// TIA Portal V20 export
FUNCTION_BLOCK "Sequence_2_SideTapeAttachment"   // FB32852, LAD
TITLE = Sequence
// Sequence template programmend in ladder logic
// stored: IsIECCheckEnabled true, MemoryReserve 100, Namespace Unit1.Em4, SetENOAutomatically true
   VAR_INPUT
      unitStatus { ExternalAccessible := 'False'; ExternalVisible := 'False'; ExternalWritable := 'False'} : "LAF_typeUnitStatus";   // Current unit status o be used in this EM
   END_VAR
   VAR
      instSequenceLADControl { ExternalAccessible := 'False'; ExternalVisible := 'False'; ExternalWritable := 'False'} : "LAF_ControlLadSequence";
      instSequenceLADStatus { ExternalAccessible := 'False'; ExternalVisible := 'False'; ExternalWritable := 'False'} : "LAF_StatusLadSequence";
      statTonTime { ExternalAccessible := 'False'; ExternalVisible := 'False'; ExternalWritable := 'False'} : Array[0..9999] of TON_TIME;
   END_VAR
   VAR_TEMP
      tempCustomerAction : Bool;   // Placeholder for possible actions
      tempDo_nothing_and_wait_for_init : Bool;   // Placeholder for doing nothing
      tempSafeStateCondition : Bool;   // Temp Condition for the equipment module to be in a safe state
   END_VAR
   VAR CONSTANT
      delayTime : Time := T#100ms;
      STEP_IDLE : DInt := 1;
      JOB_1_STEP_1 : DInt := 101;
      JOB_1_STEP_10 : DInt := 110;
      JOB_1_STEP_11 : DInt := 111;
      JOB_1_STEP_20 : DInt := 120;
      JOB_1_STEP_30 : DInt := 130;
      JOB_1_STEP_31 : DInt := 131;
      JOB_1_STEP_32 : DInt := 132;
      JOB_1_STEP_33 : DInt := 133;
      JOB_1_STEP_34 : DInt := 134;
      JOB_1_STEP_40 : DInt := 140;
      JOB_1_STEP_41 : DInt := 141;
      JOB_1_STEP_42 : DInt := 142;
      JOB_1_STEP_43 : DInt := 143;
      JOB_1_STEP_44 : DInt := 144;
      JOB_1_STEP_80 : DInt := 180;
      JOB_1_STEP_81 : DInt := 181;
      JOB_1_STEP_90 : DInt := 190;
      JOB_3_STEP_1 : DInt := 301;
      JOB_3_STEP_10 : DInt := 310;
      JOB_3_STEP_20 : DInt := 320;
      JOB_3_STEP_21 : DInt := 321;
      JOB_3_STEP_30 : DInt := 330;
      JOB_3_STEP_31 : DInt := 331;
      JOB_3_STEP_40 : DInt := 340;
      JOB_3_STEP_41 : DInt := 341;
      JOB_3_STEP_70 : DInt := 370;
      JOB_3_STEP_80 : DInt := 380;
      JOB_3_STEP_90 : DInt := 390;
      JOB_2_STEP_1 : DInt := 201;
      JOB_2_STEP_10 : DInt := 210;
      JOB_2_STEP_20 : DInt := 220;
      JOB_2_STEP_21 : DInt := 221;
      JOB_2_STEP_30 : DInt := 230;
      JOB_2_STEP_31 : DInt := 231;
      JOB_2_STEP_40 : DInt := 240;
      JOB_2_STEP_41 : DInt := 241;
      JOB_2_STEP_70 : DInt := 270;
      JOB_2_STEP_80 : DInt := 280;
      JOB_2_STEP_90 : DInt := 290;
      JOB_4_STEP_1 : DInt := 401;
      JOB_4_STEP_10 : DInt := 410;
      JOB_4_STEP_20 : DInt := 420;
      JOB_4_STEP_21 : DInt := 421;
      JOB_4_STEP_22 : DInt := 422;
      JOB_4_STEP_30 : DInt := 430;
      JOB_4_STEP_31 : DInt := 431;
      JOB_4_STEP_80 : DInt := 480;
      JOB_4_STEP_90 : DInt := 490;
      JOB_5_STEP_1 : DInt := 501;
      JOB_5_STEP_10 : DInt := 510;
      JOB_5_STEP_20 : DInt := 520;
      JOB_5_STEP_21 : DInt := 521;
      JOB_5_STEP_22 : DInt := 522;
      JOB_5_STEP_30 : DInt := 530;
      JOB_5_STEP_31 : DInt := 531;
      JOB_5_STEP_80 : DInt := 580;
      JOB_5_STEP_90 : DInt := 590;
      JOB_6_STEP_1 : DInt := 601;
      JOB_6_STEP_10 : DInt := 610;
      JOB_6_STEP_20 : DInt := 620;
      JOB_6_STEP_21 : DInt := 621;
      JOB_6_STEP_22 : DInt := 622;
      JOB_6_STEP_30 : DInt := 630;
      JOB_6_STEP_31 : DInt := 631;
      JOB_6_STEP_80 : DInt := 680;
      JOB_6_STEP_90 : DInt := 690;
      JOB_7_STEP_1 : DInt := 701;
      JOB_7_STEP_10 : DInt := 710;
      JOB_7_STEP_20 : DInt := 720;
      JOB_7_STEP_21 : DInt := 721;
      JOB_7_STEP_22 : DInt := 722;
      JOB_7_STEP_30 : DInt := 730;
      JOB_7_STEP_31 : DInt := 731;
      JOB_7_STEP_80 : DInt := 780;
      JOB_7_STEP_90 : DInt := 790;
      JOB_8_STEP_1 : DInt := 801;
      JOB_8_STEP_10 : DInt := 810;
      JOB_8_STEP_11 : DInt := 811;
      JOB_8_STEP_12 : DInt := 812;
      JOB_8_STEP_13 : DInt := 813;
      JOB_8_STEP_14 : DInt := 814;
      JOB_8_STEP_15 : DInt := 815;
      JOB_8_STEP_16 : DInt := 816;
      JOB_8_STEP_17 : DInt := 817;
      JOB_8_STEP_20 : DInt := 820;
      JOB_8_STEP_21 : DInt := 821;
      JOB_8_STEP_22 : DInt := 822;
      JOB_8_STEP_23 : DInt := 823;
      JOB_8_STEP_24 : DInt := 824;
      JOB_8_STEP_25 : DInt := 825;
      JOB_8_STEP_26 : DInt := 826;
      JOB_8_STEP_27 : DInt := 827;
      JOB_8_STEP_30 : DInt := 830;
      JOB_8_STEP_31 : DInt := 831;
      JOB_8_STEP_60 : DInt := 860;
      JOB_8_STEP_70 : DInt := 880;
      JOB_8_STEP_80 : DInt := 890;
      STEP_IMMEDIATE_STOP : DInt := 9001;   // Step executed when an immediate stop command is triggered for the sequence (i.e. when unit is in state aborting)
      TO_DO_INSERT_ACTIONS_HERE : Bool := TRUE;   // Template : Add actions
      TO_DO_INSERT_CONDITION_FOR_TRANSITION_HERE : Bool := TRUE;   // Template : Add conditions
   END_VAR
   VAR_TEMP   // added for the SCL form of the ladder/FBD networks
      _w1 : Bool;
      _w2 : Bool;
   END_VAR
BEGIN

REGION Network 1: BLOCK INFO HEADER
   // (company) / (C) Copyright (year)
   // ---------------------------------------------------------------------------------
   // Title:                             (Title of this block)
   // Comment/Function: (that is implemented in the block)
   // Library/Family:           (that the source is dedicated to)
   // Author:                        (department / person in charge / contact)
   // Target System:          (test system with FW version)
   // Engineering:              TIA Portal (SW version)
   // Restrictions:               (OB types, etc.)
   // Requirements:           (hardware, technological package, etc.)
   // ---------------------------------------------------------------------------------
   // Change log table:
   // Version          | Date             | Signature      | Expert in charge  | Changes applied ------------------------|----------------------|-------------------------|--------------------------------|-----------------------
   // 001.000.000 | yyyy-mm-dd | 0x00000000 | (name of expert) | First released version
END_REGION

REGION Network 2: DESCRIPTION
   // This is a template block provided by the Automation Framework. It can be used to create an own project.
   // The Block Info Header is prepared to put in your own data.
   // Description of the block could be added here and the docu created by Code2Docu.
END_REGION

REGION Network 3: *************** CONTROL **********************
END_REGION

REGION Network 4: Sequence Control ("Enter your Sequins number here")
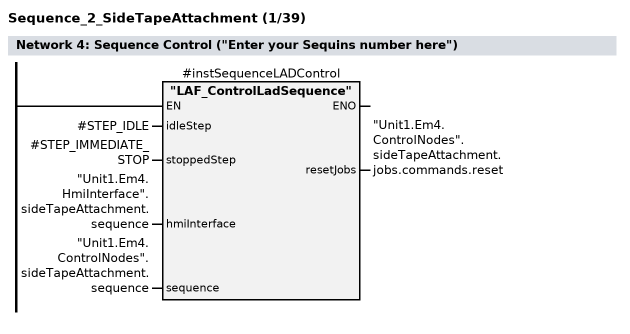
   RUNG wire#powerrail
      #instSequenceLADControl(idleStep := #STEP_IDLE, stoppedStep := #STEP_IMMEDIATE_STOP, hmiInterface := "Unit1.Em4.HmiInterface".sideTapeAttachment.sequence, sequence := "Unit1.Em4.ControlNodes".sideTapeAttachment.sequence, resetJobs => "Unit1.Em4.ControlNodes".sideTapeAttachment.jobs.commands.reset)
   END_RUNG
   // the same network as SCL:
   #instSequenceLADControl(idleStep := #STEP_IDLE,   // "LAF_ControlLadSequence"
                           stoppedStep := #STEP_IMMEDIATE_STOP,
                           hmiInterface := "Unit1.Em4.HmiInterface".sideTapeAttachment.sequence,
                           sequence := "Unit1.Em4.ControlNodes".sideTapeAttachment.sequence,
                           resetJobs => "Unit1.Em4.ControlNodes".sideTapeAttachment.jobs.commands.reset);
END_REGION

REGION Network 5: Step IDLE
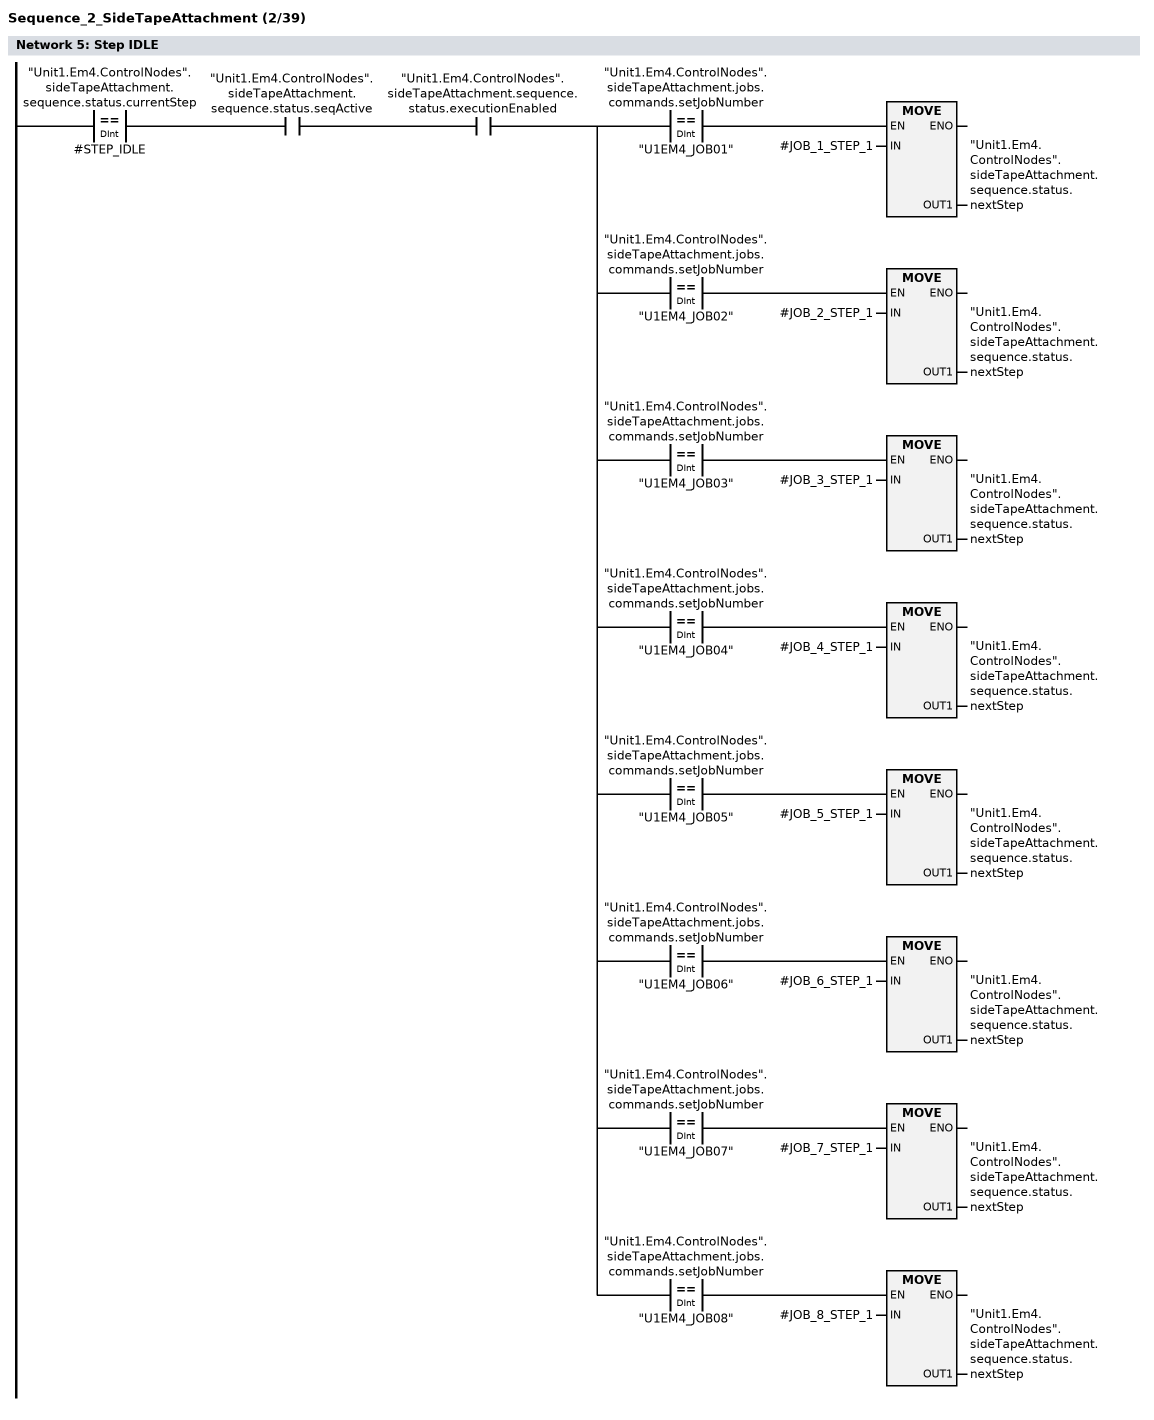
   RUNG wire#powerrail
      { S7_Templates := "SrcType := DInt" } EQ_Contact(in1 := "Unit1.Em4.ControlNodes".sideTapeAttachment.sequence.status.currentStep, in2 := #STEP_IDLE)
      Contact( "Unit1.Em4.ControlNodes".sideTapeAttachment.sequence.status.seqActive )
      Contact( "Unit1.Em4.ControlNodes".sideTapeAttachment.sequence.status.executionEnabled )
      wire#w1
      { S7_Templates := "SrcType := DInt" } EQ_Contact(in1 := "Unit1.Em4.ControlNodes".sideTapeAttachment.jobs.commands.setJobNumber, in2 := "U1EM4_JOB01")
      Move(in := #JOB_1_STEP_1, out1 => "Unit1.Em4.ControlNodes".sideTapeAttachment.sequence.status.nextStep)
   END_RUNG
   RUNG wire#w1
      { S7_Templates := "SrcType := DInt" } EQ_Contact(in1 := "Unit1.Em4.ControlNodes".sideTapeAttachment.jobs.commands.setJobNumber, in2 := "U1EM4_JOB02")
      Move(in := #JOB_2_STEP_1, out1 => "Unit1.Em4.ControlNodes".sideTapeAttachment.sequence.status.nextStep)
   END_RUNG
   RUNG wire#w1
      { S7_Templates := "SrcType := DInt" } EQ_Contact(in1 := "Unit1.Em4.ControlNodes".sideTapeAttachment.jobs.commands.setJobNumber, in2 := "U1EM4_JOB03")
      Move(in := #JOB_3_STEP_1, out1 => "Unit1.Em4.ControlNodes".sideTapeAttachment.sequence.status.nextStep)
   END_RUNG
   RUNG wire#w1
      { S7_Templates := "SrcType := DInt" } EQ_Contact(in1 := "Unit1.Em4.ControlNodes".sideTapeAttachment.jobs.commands.setJobNumber, in2 := "U1EM4_JOB04")
      Move(in := #JOB_4_STEP_1, out1 => "Unit1.Em4.ControlNodes".sideTapeAttachment.sequence.status.nextStep)
   END_RUNG
   RUNG wire#w1
      { S7_Templates := "SrcType := DInt" } EQ_Contact(in1 := "Unit1.Em4.ControlNodes".sideTapeAttachment.jobs.commands.setJobNumber, in2 := "U1EM4_JOB05")
      Move(in := #JOB_5_STEP_1, out1 => "Unit1.Em4.ControlNodes".sideTapeAttachment.sequence.status.nextStep)
   END_RUNG
   RUNG wire#w1
      { S7_Templates := "SrcType := DInt" } EQ_Contact(in1 := "Unit1.Em4.ControlNodes".sideTapeAttachment.jobs.commands.setJobNumber, in2 := "U1EM4_JOB06")
      Move(in := #JOB_6_STEP_1, out1 => "Unit1.Em4.ControlNodes".sideTapeAttachment.sequence.status.nextStep)
   END_RUNG
   RUNG wire#w1
      { S7_Templates := "SrcType := DInt" } EQ_Contact(in1 := "Unit1.Em4.ControlNodes".sideTapeAttachment.jobs.commands.setJobNumber, in2 := "U1EM4_JOB07")
      Move(in := #JOB_7_STEP_1, out1 => "Unit1.Em4.ControlNodes".sideTapeAttachment.sequence.status.nextStep)
   END_RUNG
   RUNG wire#w1
      { S7_Templates := "SrcType := DInt" } EQ_Contact(in1 := "Unit1.Em4.ControlNodes".sideTapeAttachment.jobs.commands.setJobNumber, in2 := "U1EM4_JOB08")
      Move(in := #JOB_8_STEP_1, out1 => "Unit1.Em4.ControlNodes".sideTapeAttachment.sequence.status.nextStep)
   END_RUNG
   // the same network as SCL:
   #_w1 := ("Unit1.Em4.ControlNodes".sideTapeAttachment.sequence.status.currentStep = #STEP_IDLE) AND "Unit1.Em4.ControlNodes".sideTapeAttachment.sequence.status.seqActive AND "Unit1.Em4.ControlNodes".sideTapeAttachment.sequence.status.executionEnabled;
   IF #_w1 AND ("Unit1.Em4.ControlNodes".sideTapeAttachment.jobs.commands.setJobNumber = "U1EM4_JOB01") THEN
       "Unit1.Em4.ControlNodes".sideTapeAttachment.sequence.status.nextStep := #JOB_1_STEP_1;
   END_IF;
   IF #_w1 AND ("Unit1.Em4.ControlNodes".sideTapeAttachment.jobs.commands.setJobNumber = "U1EM4_JOB02") THEN
       "Unit1.Em4.ControlNodes".sideTapeAttachment.sequence.status.nextStep := #JOB_2_STEP_1;
   END_IF;
   IF #_w1 AND ("Unit1.Em4.ControlNodes".sideTapeAttachment.jobs.commands.setJobNumber = "U1EM4_JOB03") THEN
       "Unit1.Em4.ControlNodes".sideTapeAttachment.sequence.status.nextStep := #JOB_3_STEP_1;
   END_IF;
   IF #_w1 AND ("Unit1.Em4.ControlNodes".sideTapeAttachment.jobs.commands.setJobNumber = "U1EM4_JOB04") THEN
       "Unit1.Em4.ControlNodes".sideTapeAttachment.sequence.status.nextStep := #JOB_4_STEP_1;
   END_IF;
   IF #_w1 AND ("Unit1.Em4.ControlNodes".sideTapeAttachment.jobs.commands.setJobNumber = "U1EM4_JOB05") THEN
       "Unit1.Em4.ControlNodes".sideTapeAttachment.sequence.status.nextStep := #JOB_5_STEP_1;
   END_IF;
   IF #_w1 AND ("Unit1.Em4.ControlNodes".sideTapeAttachment.jobs.commands.setJobNumber = "U1EM4_JOB06") THEN
       "Unit1.Em4.ControlNodes".sideTapeAttachment.sequence.status.nextStep := #JOB_6_STEP_1;
   END_IF;
   IF #_w1 AND ("Unit1.Em4.ControlNodes".sideTapeAttachment.jobs.commands.setJobNumber = "U1EM4_JOB07") THEN
       "Unit1.Em4.ControlNodes".sideTapeAttachment.sequence.status.nextStep := #JOB_7_STEP_1;
   END_IF;
   IF #_w1 AND ("Unit1.Em4.ControlNodes".sideTapeAttachment.jobs.commands.setJobNumber = "U1EM4_JOB08") THEN
       "Unit1.Em4.ControlNodes".sideTapeAttachment.sequence.status.nextStep := #JOB_8_STEP_1;
   END_IF;
END_REGION

REGION Network 6: ******************** JOB[1] EM HOMING ********************
END_REGION

REGION Network 7: Step[101] : JOB[1] Condition
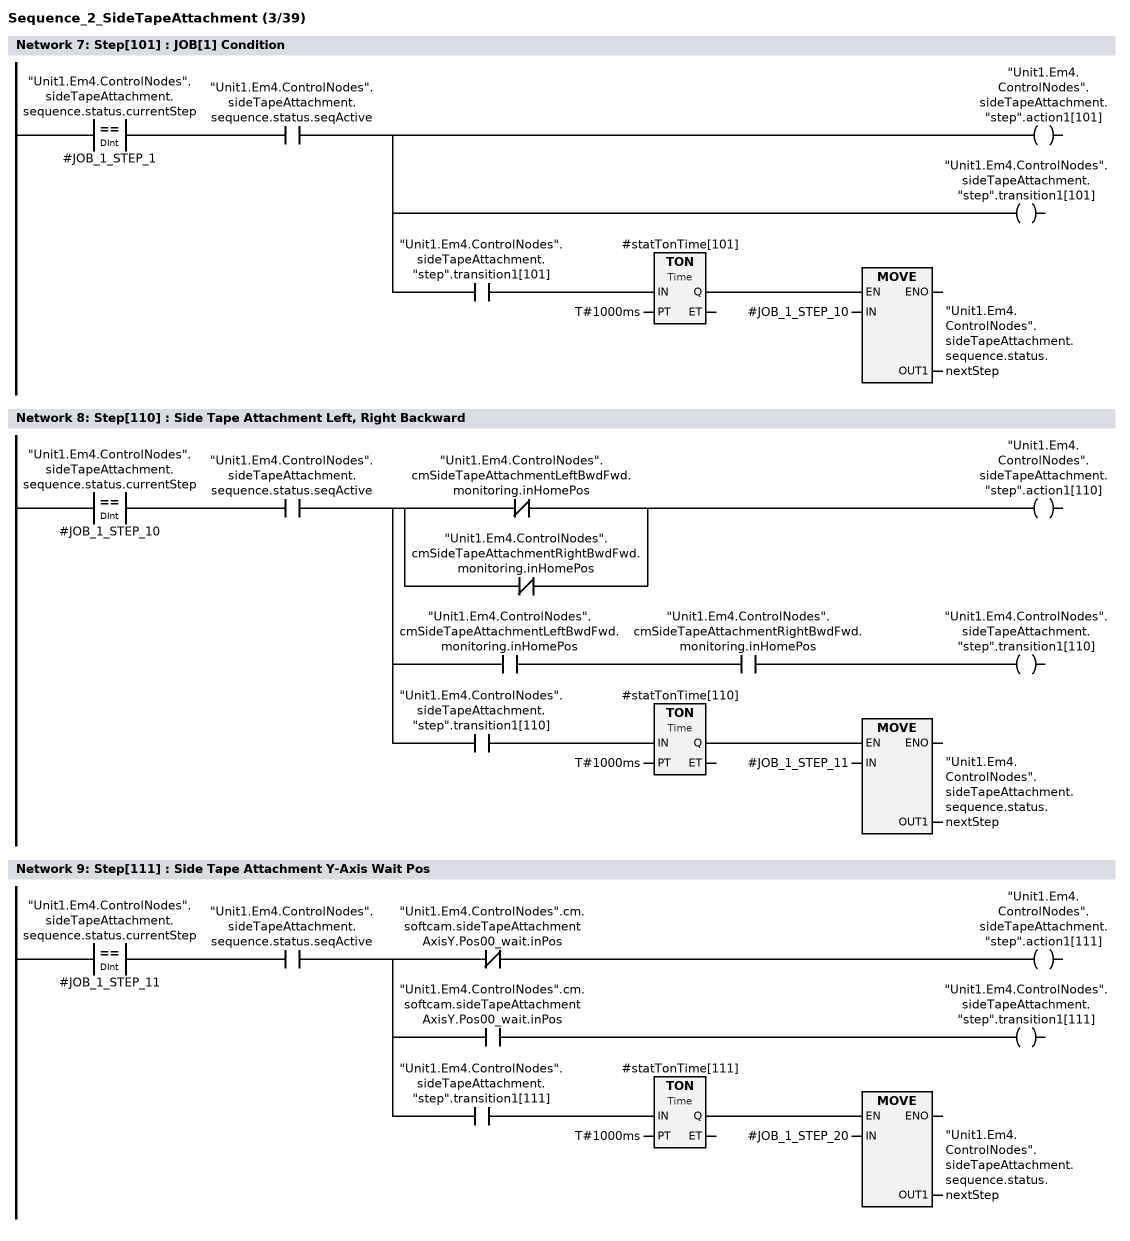
   RUNG wire#powerrail
      { S7_Templates := "SrcType := DInt" } EQ_Contact(in1 := "Unit1.Em4.ControlNodes".sideTapeAttachment.sequence.status.currentStep, in2 := #JOB_1_STEP_1)
      Contact( "Unit1.Em4.ControlNodes".sideTapeAttachment.sequence.status.seqActive )
      wire#w1
      Coil( "Unit1.Em4.ControlNodes".sideTapeAttachment."step".action1[101] )
   END_RUNG
   RUNG wire#w1
      Coil( "Unit1.Em4.ControlNodes".sideTapeAttachment."step".transition1[101] )
   END_RUNG
   RUNG wire#w1
      Contact( "Unit1.Em4.ControlNodes".sideTapeAttachment."step".transition1[101] )
      { S7_Templates := "time_type := Time" } #statTonTime[101].TON(pt := T#1000ms, et =>)
      Move(in := #JOB_1_STEP_10, out1 => "Unit1.Em4.ControlNodes".sideTapeAttachment.sequence.status.nextStep)
   END_RUNG
   // the same network as SCL:
   "Unit1.Em4.ControlNodes".sideTapeAttachment."step".action1[101] := ("Unit1.Em4.ControlNodes".sideTapeAttachment.sequence.status.currentStep = #JOB_1_STEP_1) AND "Unit1.Em4.ControlNodes".sideTapeAttachment.sequence.status.seqActive;
   "Unit1.Em4.ControlNodes".sideTapeAttachment."step".transition1[101] := ("Unit1.Em4.ControlNodes".sideTapeAttachment.sequence.status.currentStep = #JOB_1_STEP_1) AND "Unit1.Em4.ControlNodes".sideTapeAttachment.sequence.status.seqActive;
   #statTonTime[101].TON(IN := ("Unit1.Em4.ControlNodes".sideTapeAttachment.sequence.status.currentStep = #JOB_1_STEP_1) AND "Unit1.Em4.ControlNodes".sideTapeAttachment.sequence.status.seqActive AND "Unit1.Em4.ControlNodes".sideTapeAttachment."step".transition1[101],
                         PT := T#1000ms);
   IF #statTonTime[101].Q THEN
       "Unit1.Em4.ControlNodes".sideTapeAttachment.sequence.status.nextStep := #JOB_1_STEP_10;
   END_IF;
END_REGION

REGION Network 8: Step[110] : Side Tape Attachment Left, Right Backward
   RUNG wire#powerrail
      { S7_Templates := "SrcType := DInt" } EQ_Contact(in1 := "Unit1.Em4.ControlNodes".sideTapeAttachment.sequence.status.currentStep, in2 := #JOB_1_STEP_10)
      Contact( "Unit1.Em4.ControlNodes".sideTapeAttachment.sequence.status.seqActive )
      wire#w1
      I_Contact( "Unit1.Em4.ControlNodes".cmSideTapeAttachmentLeftBwdFwd.monitoring.inHomePos )
      wire#w2
      Coil( "Unit1.Em4.ControlNodes".sideTapeAttachment."step".action1[110] )
   END_RUNG
   RUNG wire#w1
      I_Contact( "Unit1.Em4.ControlNodes".cmSideTapeAttachmentRightBwdFwd.monitoring.inHomePos )
   END_RUNG wire#w2
   RUNG wire#w1
      Contact( "Unit1.Em4.ControlNodes".cmSideTapeAttachmentLeftBwdFwd.monitoring.inHomePos )
      Contact( "Unit1.Em4.ControlNodes".cmSideTapeAttachmentRightBwdFwd.monitoring.inHomePos )
      Coil( "Unit1.Em4.ControlNodes".sideTapeAttachment."step".transition1[110] )
   END_RUNG
   RUNG wire#w1
      Contact( "Unit1.Em4.ControlNodes".sideTapeAttachment."step".transition1[110] )
      { S7_Templates := "time_type := Time" } #statTonTime[110].TON(pt := T#1000ms, et =>)
      Move(in := #JOB_1_STEP_11, out1 => "Unit1.Em4.ControlNodes".sideTapeAttachment.sequence.status.nextStep)
   END_RUNG
   // the same network as SCL:
   #_w1 := ("Unit1.Em4.ControlNodes".sideTapeAttachment.sequence.status.currentStep = #JOB_1_STEP_10) AND "Unit1.Em4.ControlNodes".sideTapeAttachment.sequence.status.seqActive;
   "Unit1.Em4.ControlNodes".sideTapeAttachment."step".action1[110] := #_w1 AND (NOT "Unit1.Em4.ControlNodes".cmSideTapeAttachmentLeftBwdFwd.monitoring.inHomePos OR NOT "Unit1.Em4.ControlNodes".cmSideTapeAttachmentRightBwdFwd.monitoring.inHomePos);
   "Unit1.Em4.ControlNodes".sideTapeAttachment."step".transition1[110] := #_w1 AND "Unit1.Em4.ControlNodes".cmSideTapeAttachmentLeftBwdFwd.monitoring.inHomePos AND "Unit1.Em4.ControlNodes".cmSideTapeAttachmentRightBwdFwd.monitoring.inHomePos;
   #statTonTime[110].TON(IN := #_w1 AND "Unit1.Em4.ControlNodes".sideTapeAttachment."step".transition1[110],
                         PT := T#1000ms);
   IF #statTonTime[110].Q THEN
       "Unit1.Em4.ControlNodes".sideTapeAttachment.sequence.status.nextStep := #JOB_1_STEP_11;
   END_IF;
END_REGION

REGION Network 9: Step[111] : Side Tape Attachment Y-Axis Wait Pos
   RUNG wire#powerrail
      { S7_Templates := "SrcType := DInt" } EQ_Contact(in1 := "Unit1.Em4.ControlNodes".sideTapeAttachment.sequence.status.currentStep, in2 := #JOB_1_STEP_11)
      Contact( "Unit1.Em4.ControlNodes".sideTapeAttachment.sequence.status.seqActive )
      wire#w1
      I_Contact( "Unit1.Em4.ControlNodes".cm.softcam.sideTapeAttachmentAxisY.Pos00_wait.inPos )
      Coil( "Unit1.Em4.ControlNodes".sideTapeAttachment."step".action1[111] )
   END_RUNG
   RUNG wire#w1
      Contact( "Unit1.Em4.ControlNodes".cm.softcam.sideTapeAttachmentAxisY.Pos00_wait.inPos )
      Coil( "Unit1.Em4.ControlNodes".sideTapeAttachment."step".transition1[111] )
   END_RUNG
   RUNG wire#w1
      Contact( "Unit1.Em4.ControlNodes".sideTapeAttachment."step".transition1[111] )
      { S7_Templates := "time_type := Time" } #statTonTime[111].TON(pt := T#1000ms, et =>)
      Move(in := #JOB_1_STEP_20, out1 => "Unit1.Em4.ControlNodes".sideTapeAttachment.sequence.status.nextStep)
   END_RUNG
   // the same network as SCL:
   #_w1 := ("Unit1.Em4.ControlNodes".sideTapeAttachment.sequence.status.currentStep = #JOB_1_STEP_11) AND "Unit1.Em4.ControlNodes".sideTapeAttachment.sequence.status.seqActive;
   "Unit1.Em4.ControlNodes".sideTapeAttachment."step".action1[111] := #_w1 AND NOT "Unit1.Em4.ControlNodes".cm.softcam.sideTapeAttachmentAxisY.Pos00_wait.inPos;
   "Unit1.Em4.ControlNodes".sideTapeAttachment."step".transition1[111] := #_w1 AND "Unit1.Em4.ControlNodes".cm.softcam.sideTapeAttachmentAxisY.Pos00_wait.inPos;
   #statTonTime[111].TON(IN := #_w1 AND "Unit1.Em4.ControlNodes".sideTapeAttachment."step".transition1[111],
                         PT := T#1000ms);
   IF #statTonTime[111].Q THEN
       "Unit1.Em4.ControlNodes".sideTapeAttachment.sequence.status.nextStep := #JOB_1_STEP_20;
   END_IF;
END_REGION

REGION Network 10: Step[120] : Side Tape Attachment Bottom Forward
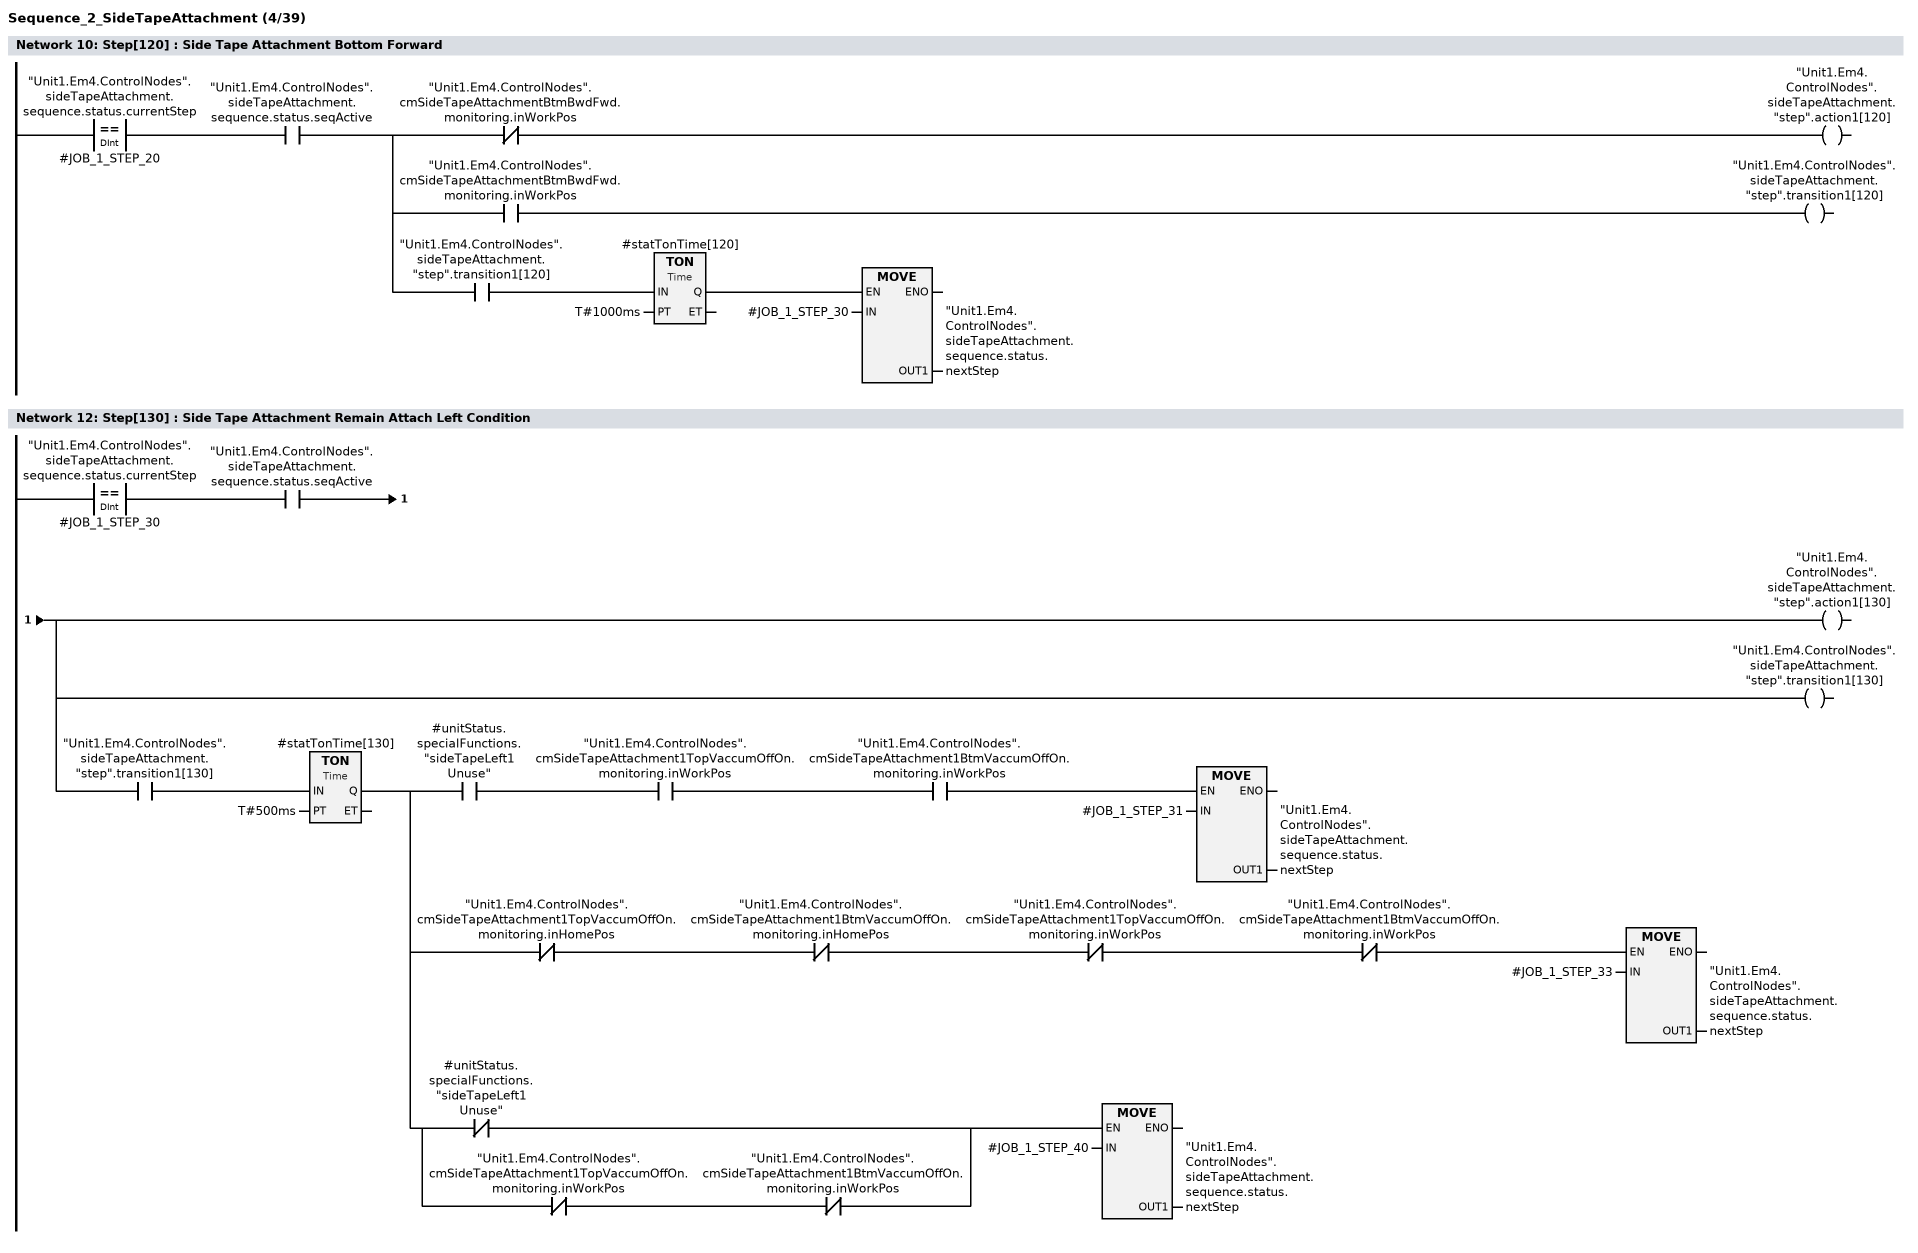
   RUNG wire#powerrail
      { S7_Templates := "SrcType := DInt" } EQ_Contact(in1 := "Unit1.Em4.ControlNodes".sideTapeAttachment.sequence.status.currentStep, in2 := #JOB_1_STEP_20)
      Contact( "Unit1.Em4.ControlNodes".sideTapeAttachment.sequence.status.seqActive )
      wire#w1
      I_Contact( "Unit1.Em4.ControlNodes".cmSideTapeAttachmentBtmBwdFwd.monitoring.inWorkPos )
      Coil( "Unit1.Em4.ControlNodes".sideTapeAttachment."step".action1[120] )
   END_RUNG
   RUNG wire#w1
      Contact( "Unit1.Em4.ControlNodes".cmSideTapeAttachmentBtmBwdFwd.monitoring.inWorkPos )
      Coil( "Unit1.Em4.ControlNodes".sideTapeAttachment."step".transition1[120] )
   END_RUNG
   RUNG wire#w1
      Contact( "Unit1.Em4.ControlNodes".sideTapeAttachment."step".transition1[120] )
      { S7_Templates := "time_type := Time" } #statTonTime[120].TON(pt := T#1000ms, et =>)
      Move(in := #JOB_1_STEP_30, out1 => "Unit1.Em4.ControlNodes".sideTapeAttachment.sequence.status.nextStep)
   END_RUNG
   // the same network as SCL:
   #_w1 := ("Unit1.Em4.ControlNodes".sideTapeAttachment.sequence.status.currentStep = #JOB_1_STEP_20) AND "Unit1.Em4.ControlNodes".sideTapeAttachment.sequence.status.seqActive;
   "Unit1.Em4.ControlNodes".sideTapeAttachment."step".action1[120] := #_w1 AND NOT "Unit1.Em4.ControlNodes".cmSideTapeAttachmentBtmBwdFwd.monitoring.inWorkPos;
   "Unit1.Em4.ControlNodes".sideTapeAttachment."step".transition1[120] := #_w1 AND "Unit1.Em4.ControlNodes".cmSideTapeAttachmentBtmBwdFwd.monitoring.inWorkPos;
   #statTonTime[120].TON(IN := #_w1 AND "Unit1.Em4.ControlNodes".sideTapeAttachment."step".transition1[120],
                         PT := T#1000ms);
   IF #statTonTime[120].Q THEN
       "Unit1.Em4.ControlNodes".sideTapeAttachment.sequence.status.nextStep := #JOB_1_STEP_30;
   END_IF;
END_REGION

REGION Network 11: ******************** STEP[130~134] SIDE TAPE ATTACHMENT LEFT REMAIN ATTACH ********************
END_REGION

REGION Network 12: Step[130] : Side Tape Attachment Remain Attach Left Condition
   RUNG wire#powerrail
      { S7_Templates := "SrcType := DInt" } EQ_Contact(in1 := "Unit1.Em4.ControlNodes".sideTapeAttachment.sequence.status.currentStep, in2 := #JOB_1_STEP_30)
      Contact( "Unit1.Em4.ControlNodes".sideTapeAttachment.sequence.status.seqActive )
      wire#w1
      Coil( "Unit1.Em4.ControlNodes".sideTapeAttachment."step".action1[130] )
   END_RUNG
   RUNG wire#w1
      Coil( "Unit1.Em4.ControlNodes".sideTapeAttachment."step".transition1[130] )
   END_RUNG
   RUNG wire#w1
      Contact( "Unit1.Em4.ControlNodes".sideTapeAttachment."step".transition1[130] )
      { S7_Templates := "time_type := Time" } #statTonTime[130].TON(pt := T#500ms, et =>)
      wire#w2
      Contact( #unitStatus.specialFunctions."sideTapeLeft1 Unuse" )
      Contact( "Unit1.Em4.ControlNodes".cmSideTapeAttachment1TopVaccumOffOn.monitoring.inWorkPos )
      Contact( "Unit1.Em4.ControlNodes".cmSideTapeAttachment1BtmVaccumOffOn.monitoring.inWorkPos )
      Move(in := #JOB_1_STEP_31, out1 => "Unit1.Em4.ControlNodes".sideTapeAttachment.sequence.status.nextStep)
   END_RUNG
   RUNG wire#w2
      I_Contact( "Unit1.Em4.ControlNodes".cmSideTapeAttachment1TopVaccumOffOn.monitoring.inHomePos )
      I_Contact( "Unit1.Em4.ControlNodes".cmSideTapeAttachment1BtmVaccumOffOn.monitoring.inHomePos )
      I_Contact( "Unit1.Em4.ControlNodes".cmSideTapeAttachment1TopVaccumOffOn.monitoring.inWorkPos )
      I_Contact( "Unit1.Em4.ControlNodes".cmSideTapeAttachment1BtmVaccumOffOn.monitoring.inWorkPos )
      Move(in := #JOB_1_STEP_33, out1 => "Unit1.Em4.ControlNodes".sideTapeAttachment.sequence.status.nextStep)
   END_RUNG
   RUNG wire#w2
      I_Contact( #unitStatus.specialFunctions."sideTapeLeft1 Unuse" )
      wire#w3
      Move(in := #JOB_1_STEP_40, out1 => "Unit1.Em4.ControlNodes".sideTapeAttachment.sequence.status.nextStep)
   END_RUNG
   RUNG wire#w2
      I_Contact( "Unit1.Em4.ControlNodes".cmSideTapeAttachment1TopVaccumOffOn.monitoring.inWorkPos )
      I_Contact( "Unit1.Em4.ControlNodes".cmSideTapeAttachment1BtmVaccumOffOn.monitoring.inWorkPos )
   END_RUNG wire#w3
   // the same network as SCL:
   "Unit1.Em4.ControlNodes".sideTapeAttachment."step".action1[130] := ("Unit1.Em4.ControlNodes".sideTapeAttachment.sequence.status.currentStep = #JOB_1_STEP_30) AND "Unit1.Em4.ControlNodes".sideTapeAttachment.sequence.status.seqActive;
   "Unit1.Em4.ControlNodes".sideTapeAttachment."step".transition1[130] := ("Unit1.Em4.ControlNodes".sideTapeAttachment.sequence.status.currentStep = #JOB_1_STEP_30) AND "Unit1.Em4.ControlNodes".sideTapeAttachment.sequence.status.seqActive;
   #statTonTime[130].TON(IN := ("Unit1.Em4.ControlNodes".sideTapeAttachment.sequence.status.currentStep = #JOB_1_STEP_30) AND "Unit1.Em4.ControlNodes".sideTapeAttachment.sequence.status.seqActive AND "Unit1.Em4.ControlNodes".sideTapeAttachment."step".transition1[130],
                         PT := T#500ms);
   IF #statTonTime[130].Q AND #unitStatus.specialFunctions."sideTapeLeft1 Unuse" AND "Unit1.Em4.ControlNodes".cmSideTapeAttachment1TopVaccumOffOn.monitoring.inWorkPos AND "Unit1.Em4.ControlNodes".cmSideTapeAttachment1BtmVaccumOffOn.monitoring.inWorkPos THEN
       "Unit1.Em4.ControlNodes".sideTapeAttachment.sequence.status.nextStep := #JOB_1_STEP_31;
   END_IF;
   IF #statTonTime[130].Q AND NOT "Unit1.Em4.ControlNodes".cmSideTapeAttachment1TopVaccumOffOn.monitoring.inHomePos AND NOT "Unit1.Em4.ControlNodes".cmSideTapeAttachment1BtmVaccumOffOn.monitoring.inHomePos AND NOT "Unit1.Em4.ControlNodes".cmSideTapeAttachment1TopVaccumOffOn.monitoring.inWorkPos AND NOT "Unit1.Em4.ControlNodes".cmSideTapeAttachment1BtmVaccumOffOn.monitoring.inWorkPos THEN
       "Unit1.Em4.ControlNodes".sideTapeAttachment.sequence.status.nextStep := #JOB_1_STEP_33;
   END_IF;
   IF #statTonTime[130].Q AND (NOT #unitStatus.specialFunctions."sideTapeLeft1 Unuse" OR (NOT "Unit1.Em4.ControlNodes".cmSideTapeAttachment1TopVaccumOffOn.monitoring.inWorkPos AND NOT "Unit1.Em4.ControlNodes".cmSideTapeAttachment1BtmVaccumOffOn.monitoring.inWorkPos)) THEN
       "Unit1.Em4.ControlNodes".sideTapeAttachment.sequence.status.nextStep := #JOB_1_STEP_40;
   END_IF;
END_REGION

REGION Network 13: Step[131] : Side Tape Attachment X-Axis Remain Attach Left Position
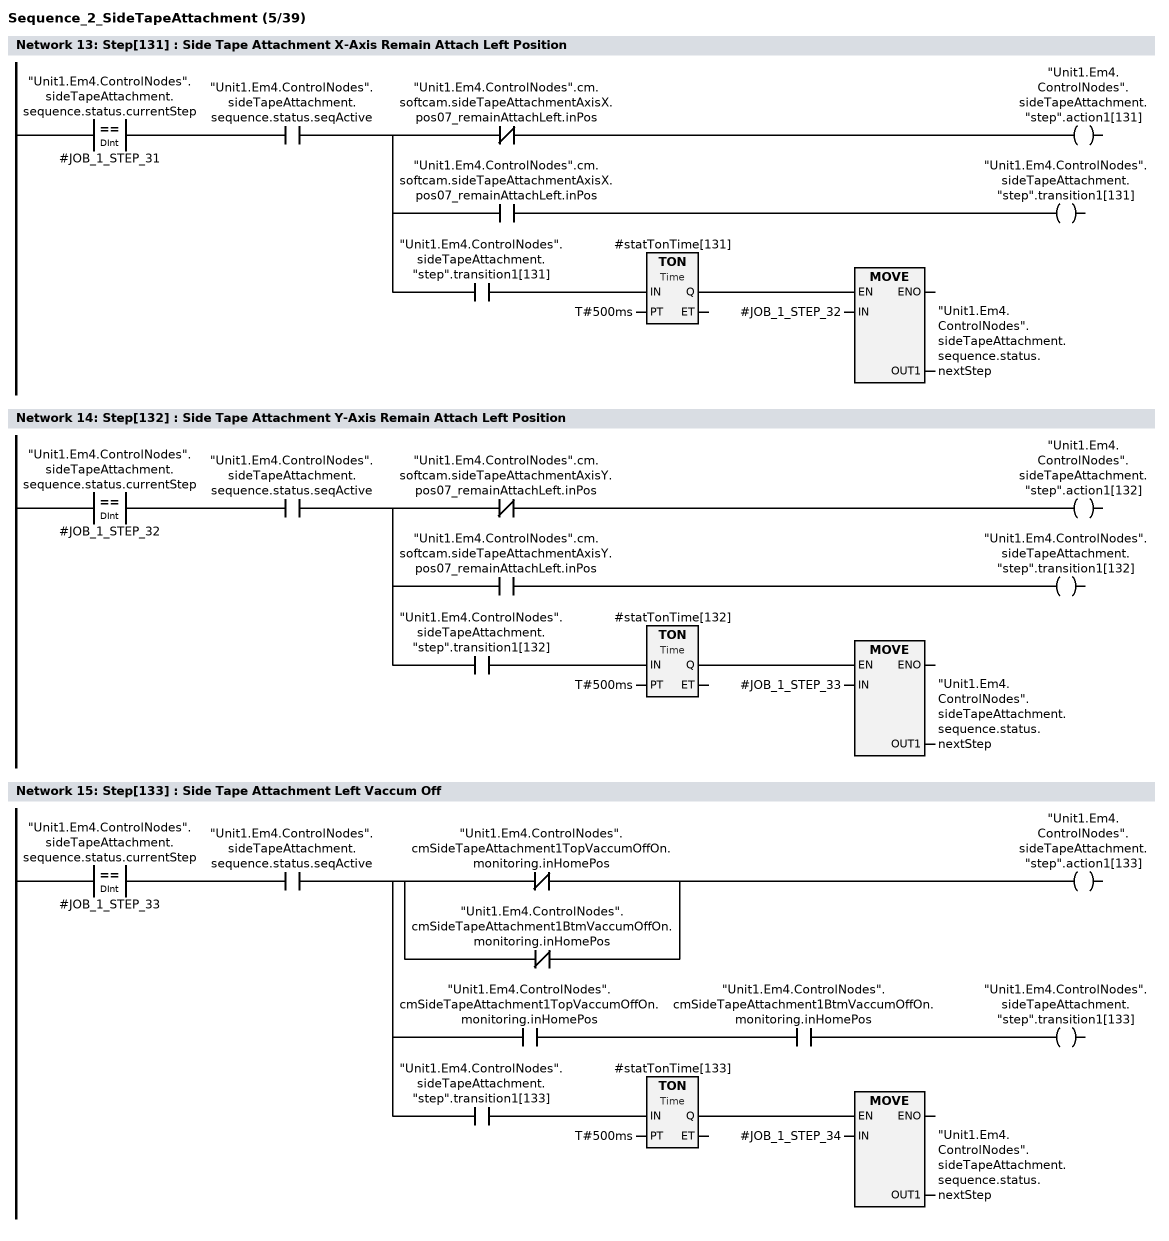
   RUNG wire#powerrail
      { S7_Templates := "SrcType := DInt" } EQ_Contact(in1 := "Unit1.Em4.ControlNodes".sideTapeAttachment.sequence.status.currentStep, in2 := #JOB_1_STEP_31)
      Contact( "Unit1.Em4.ControlNodes".sideTapeAttachment.sequence.status.seqActive )
      wire#w1
      I_Contact( "Unit1.Em4.ControlNodes".cm.softcam.sideTapeAttachmentAxisX.pos07_remainAttachLeft.inPos )
      Coil( "Unit1.Em4.ControlNodes".sideTapeAttachment."step".action1[131] )
   END_RUNG
   RUNG wire#w1
      Contact( "Unit1.Em4.ControlNodes".cm.softcam.sideTapeAttachmentAxisX.pos07_remainAttachLeft.inPos )
      Coil( "Unit1.Em4.ControlNodes".sideTapeAttachment."step".transition1[131] )
   END_RUNG
   RUNG wire#w1
      Contact( "Unit1.Em4.ControlNodes".sideTapeAttachment."step".transition1[131] )
      { S7_Templates := "time_type := Time" } #statTonTime[131].TON(pt := T#500ms, et =>)
      Move(in := #JOB_1_STEP_32, out1 => "Unit1.Em4.ControlNodes".sideTapeAttachment.sequence.status.nextStep)
   END_RUNG
   // the same network as SCL:
   #_w1 := ("Unit1.Em4.ControlNodes".sideTapeAttachment.sequence.status.currentStep = #JOB_1_STEP_31) AND "Unit1.Em4.ControlNodes".sideTapeAttachment.sequence.status.seqActive;
   "Unit1.Em4.ControlNodes".sideTapeAttachment."step".action1[131] := #_w1 AND NOT "Unit1.Em4.ControlNodes".cm.softcam.sideTapeAttachmentAxisX.pos07_remainAttachLeft.inPos;
   "Unit1.Em4.ControlNodes".sideTapeAttachment."step".transition1[131] := #_w1 AND "Unit1.Em4.ControlNodes".cm.softcam.sideTapeAttachmentAxisX.pos07_remainAttachLeft.inPos;
   #statTonTime[131].TON(IN := #_w1 AND "Unit1.Em4.ControlNodes".sideTapeAttachment."step".transition1[131],
                         PT := T#500ms);
   IF #statTonTime[131].Q THEN
       "Unit1.Em4.ControlNodes".sideTapeAttachment.sequence.status.nextStep := #JOB_1_STEP_32;
   END_IF;
END_REGION

REGION Network 14: Step[132] : Side Tape Attachment Y-Axis Remain Attach Left Position
   RUNG wire#powerrail
      { S7_Templates := "SrcType := DInt" } EQ_Contact(in1 := "Unit1.Em4.ControlNodes".sideTapeAttachment.sequence.status.currentStep, in2 := #JOB_1_STEP_32)
      Contact( "Unit1.Em4.ControlNodes".sideTapeAttachment.sequence.status.seqActive )
      wire#w1
      I_Contact( "Unit1.Em4.ControlNodes".cm.softcam.sideTapeAttachmentAxisY.pos07_remainAttachLeft.inPos )
      Coil( "Unit1.Em4.ControlNodes".sideTapeAttachment."step".action1[132] )
   END_RUNG
   RUNG wire#w1
      Contact( "Unit1.Em4.ControlNodes".cm.softcam.sideTapeAttachmentAxisY.pos07_remainAttachLeft.inPos )
      Coil( "Unit1.Em4.ControlNodes".sideTapeAttachment."step".transition1[132] )
   END_RUNG
   RUNG wire#w1
      Contact( "Unit1.Em4.ControlNodes".sideTapeAttachment."step".transition1[132] )
      { S7_Templates := "time_type := Time" } #statTonTime[132].TON(pt := T#500ms, et =>)
      Move(in := #JOB_1_STEP_33, out1 => "Unit1.Em4.ControlNodes".sideTapeAttachment.sequence.status.nextStep)
   END_RUNG
   // the same network as SCL:
   #_w1 := ("Unit1.Em4.ControlNodes".sideTapeAttachment.sequence.status.currentStep = #JOB_1_STEP_32) AND "Unit1.Em4.ControlNodes".sideTapeAttachment.sequence.status.seqActive;
   "Unit1.Em4.ControlNodes".sideTapeAttachment."step".action1[132] := #_w1 AND NOT "Unit1.Em4.ControlNodes".cm.softcam.sideTapeAttachmentAxisY.pos07_remainAttachLeft.inPos;
   "Unit1.Em4.ControlNodes".sideTapeAttachment."step".transition1[132] := #_w1 AND "Unit1.Em4.ControlNodes".cm.softcam.sideTapeAttachmentAxisY.pos07_remainAttachLeft.inPos;
   #statTonTime[132].TON(IN := #_w1 AND "Unit1.Em4.ControlNodes".sideTapeAttachment."step".transition1[132],
                         PT := T#500ms);
   IF #statTonTime[132].Q THEN
       "Unit1.Em4.ControlNodes".sideTapeAttachment.sequence.status.nextStep := #JOB_1_STEP_33;
   END_IF;
END_REGION

REGION Network 15: Step[133] : Side Tape Attachment Left Vaccum Off
   RUNG wire#powerrail
      { S7_Templates := "SrcType := DInt" } EQ_Contact(in1 := "Unit1.Em4.ControlNodes".sideTapeAttachment.sequence.status.currentStep, in2 := #JOB_1_STEP_33)
      Contact( "Unit1.Em4.ControlNodes".sideTapeAttachment.sequence.status.seqActive )
      wire#w1
      I_Contact( "Unit1.Em4.ControlNodes".cmSideTapeAttachment1TopVaccumOffOn.monitoring.inHomePos )
      wire#w2
      Coil( "Unit1.Em4.ControlNodes".sideTapeAttachment."step".action1[133] )
   END_RUNG
   RUNG wire#w1
      I_Contact( "Unit1.Em4.ControlNodes".cmSideTapeAttachment1BtmVaccumOffOn.monitoring.inHomePos )
   END_RUNG wire#w2
   RUNG wire#w1
      Contact( "Unit1.Em4.ControlNodes".cmSideTapeAttachment1TopVaccumOffOn.monitoring.inHomePos )
      Contact( "Unit1.Em4.ControlNodes".cmSideTapeAttachment1BtmVaccumOffOn.monitoring.inHomePos )
      Coil( "Unit1.Em4.ControlNodes".sideTapeAttachment."step".transition1[133] )
   END_RUNG
   RUNG wire#w1
      Contact( "Unit1.Em4.ControlNodes".sideTapeAttachment."step".transition1[133] )
      { S7_Templates := "time_type := Time" } #statTonTime[133].TON(pt := T#500ms, et =>)
      Move(in := #JOB_1_STEP_34, out1 => "Unit1.Em4.ControlNodes".sideTapeAttachment.sequence.status.nextStep)
   END_RUNG
   // the same network as SCL:
   #_w1 := ("Unit1.Em4.ControlNodes".sideTapeAttachment.sequence.status.currentStep = #JOB_1_STEP_33) AND "Unit1.Em4.ControlNodes".sideTapeAttachment.sequence.status.seqActive;
   "Unit1.Em4.ControlNodes".sideTapeAttachment."step".action1[133] := #_w1 AND (NOT "Unit1.Em4.ControlNodes".cmSideTapeAttachment1TopVaccumOffOn.monitoring.inHomePos OR NOT "Unit1.Em4.ControlNodes".cmSideTapeAttachment1BtmVaccumOffOn.monitoring.inHomePos);
   "Unit1.Em4.ControlNodes".sideTapeAttachment."step".transition1[133] := #_w1 AND "Unit1.Em4.ControlNodes".cmSideTapeAttachment1TopVaccumOffOn.monitoring.inHomePos AND "Unit1.Em4.ControlNodes".cmSideTapeAttachment1BtmVaccumOffOn.monitoring.inHomePos;
   #statTonTime[133].TON(IN := #_w1 AND "Unit1.Em4.ControlNodes".sideTapeAttachment."step".transition1[133],
                         PT := T#500ms);
   IF #statTonTime[133].Q THEN
       "Unit1.Em4.ControlNodes".sideTapeAttachment.sequence.status.nextStep := #JOB_1_STEP_34;
   END_IF;
END_REGION

REGION Network 16: Step[134] : Side Tape Attachment Y-Axis Wait Pos
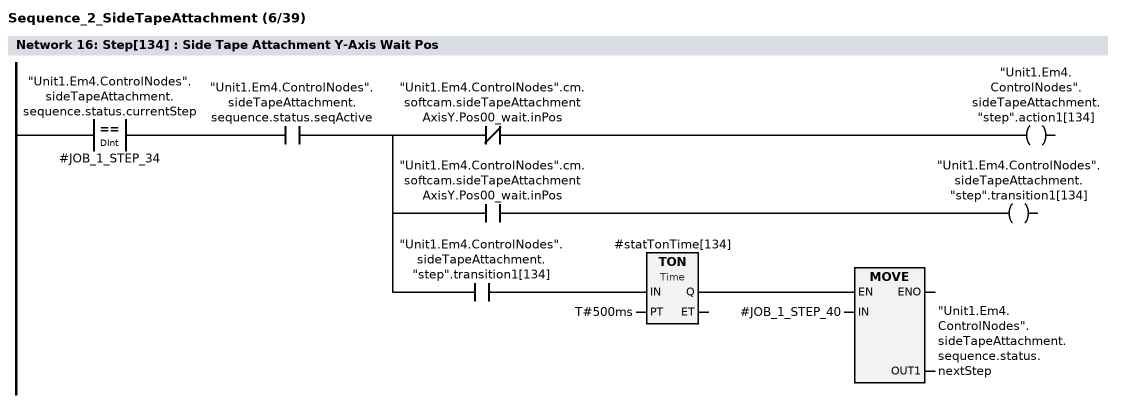
   RUNG wire#powerrail
      { S7_Templates := "SrcType := DInt" } EQ_Contact(in1 := "Unit1.Em4.ControlNodes".sideTapeAttachment.sequence.status.currentStep, in2 := #JOB_1_STEP_34)
      Contact( "Unit1.Em4.ControlNodes".sideTapeAttachment.sequence.status.seqActive )
      wire#w1
      I_Contact( "Unit1.Em4.ControlNodes".cm.softcam.sideTapeAttachmentAxisY.Pos00_wait.inPos )
      Coil( "Unit1.Em4.ControlNodes".sideTapeAttachment."step".action1[134] )
   END_RUNG
   RUNG wire#w1
      Contact( "Unit1.Em4.ControlNodes".cm.softcam.sideTapeAttachmentAxisY.Pos00_wait.inPos )
      Coil( "Unit1.Em4.ControlNodes".sideTapeAttachment."step".transition1[134] )
   END_RUNG
   RUNG wire#w1
      Contact( "Unit1.Em4.ControlNodes".sideTapeAttachment."step".transition1[134] )
      { S7_Templates := "time_type := Time" } #statTonTime[134].TON(pt := T#500ms, et =>)
      Move(in := #JOB_1_STEP_40, out1 => "Unit1.Em4.ControlNodes".sideTapeAttachment.sequence.status.nextStep)
   END_RUNG
   // the same network as SCL:
   #_w1 := ("Unit1.Em4.ControlNodes".sideTapeAttachment.sequence.status.currentStep = #JOB_1_STEP_34) AND "Unit1.Em4.ControlNodes".sideTapeAttachment.sequence.status.seqActive;
   "Unit1.Em4.ControlNodes".sideTapeAttachment."step".action1[134] := #_w1 AND NOT "Unit1.Em4.ControlNodes".cm.softcam.sideTapeAttachmentAxisY.Pos00_wait.inPos;
   "Unit1.Em4.ControlNodes".sideTapeAttachment."step".transition1[134] := #_w1 AND "Unit1.Em4.ControlNodes".cm.softcam.sideTapeAttachmentAxisY.Pos00_wait.inPos;
   #statTonTime[134].TON(IN := #_w1 AND "Unit1.Em4.ControlNodes".sideTapeAttachment."step".transition1[134],
                         PT := T#500ms);
   IF #statTonTime[134].Q THEN
       "Unit1.Em4.ControlNodes".sideTapeAttachment.sequence.status.nextStep := #JOB_1_STEP_40;
   END_IF;
END_REGION

REGION Network 17: ******************** STEP[140~144] SIDE TAPE ATTACHMENT RIGHT REMAIN ATTACH ********************
END_REGION

REGION Network 18: Step[140] : Side Tape Attachment Remain Attach Right Condition
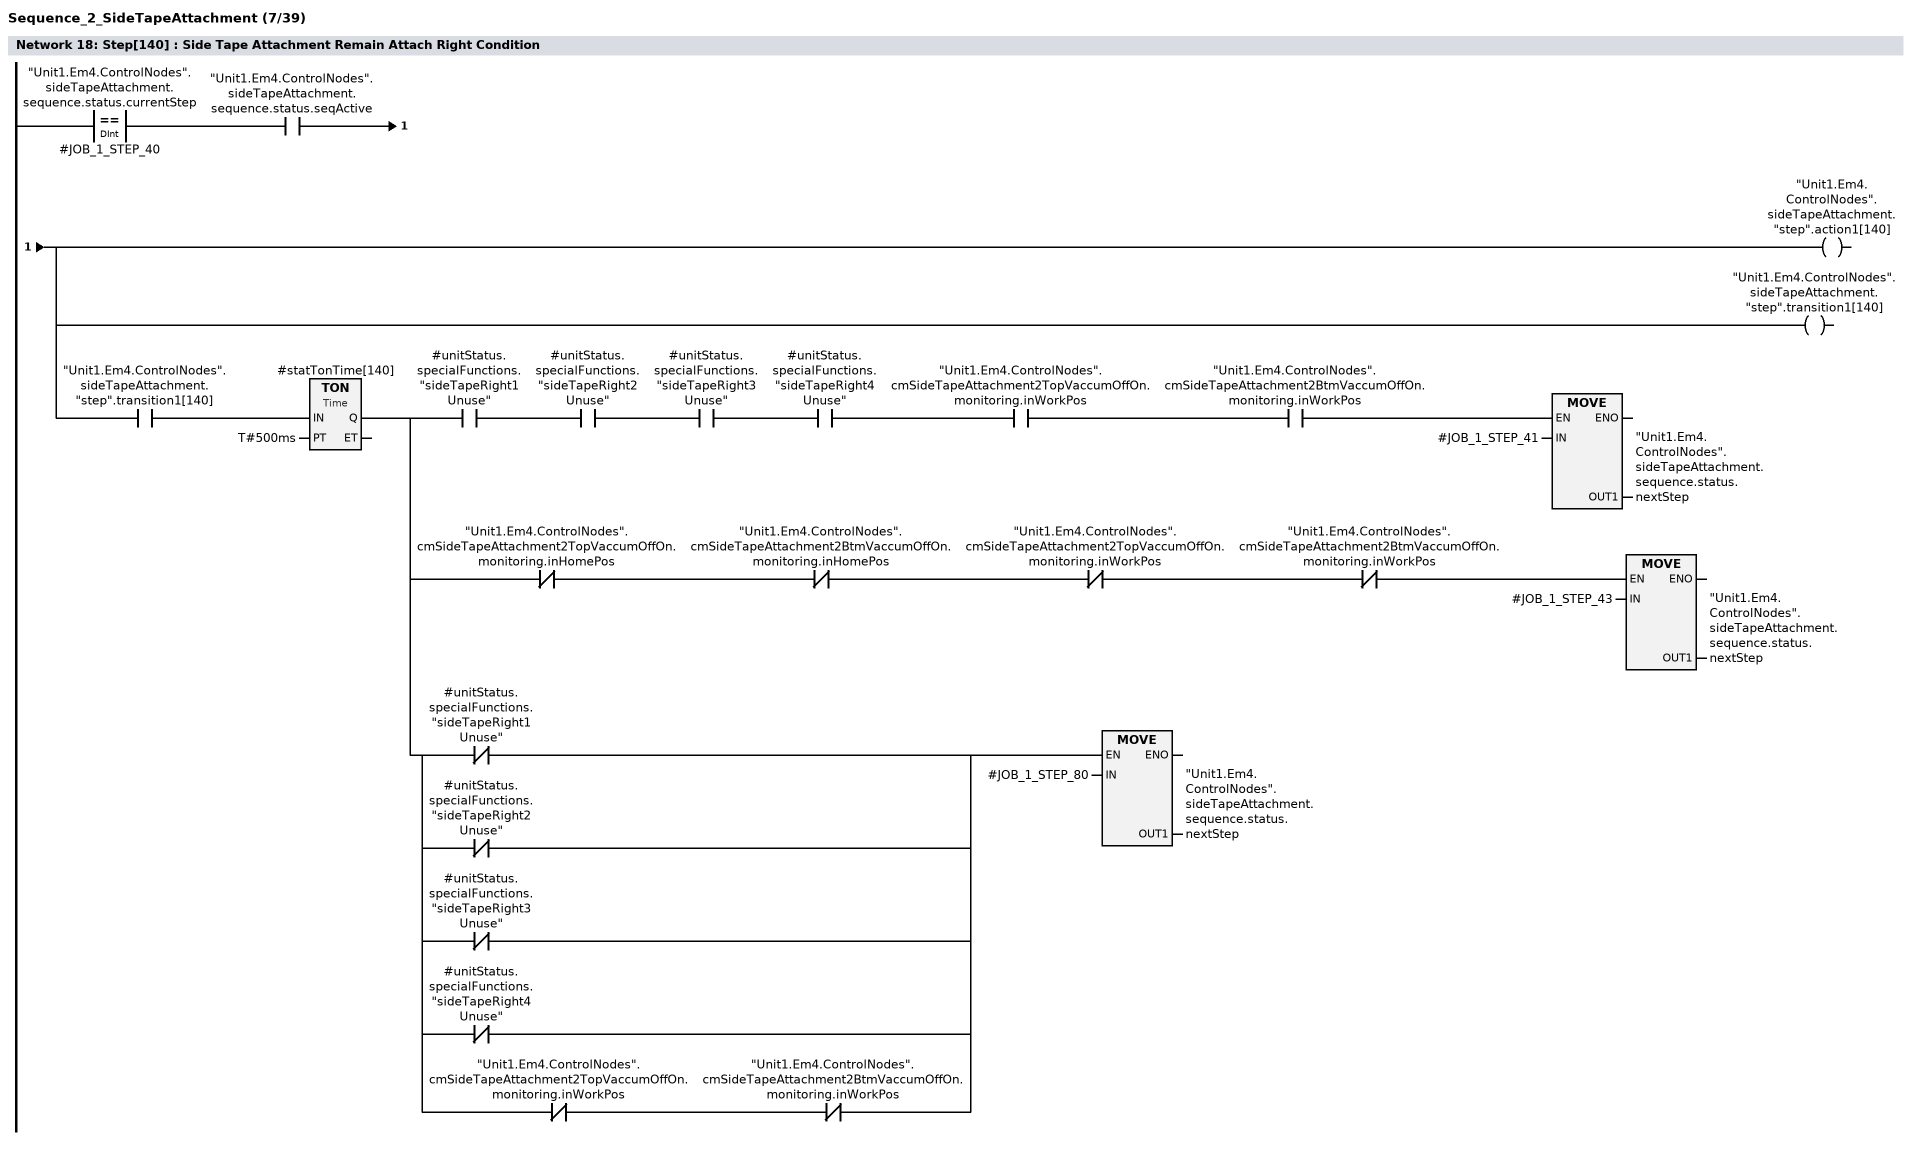
   RUNG wire#powerrail
      { S7_Templates := "SrcType := DInt" } EQ_Contact(in1 := "Unit1.Em4.ControlNodes".sideTapeAttachment.sequence.status.currentStep, in2 := #JOB_1_STEP_40)
      Contact( "Unit1.Em4.ControlNodes".sideTapeAttachment.sequence.status.seqActive )
      wire#w1
      Coil( "Unit1.Em4.ControlNodes".sideTapeAttachment."step".action1[140] )
   END_RUNG
   RUNG wire#w1
      Coil( "Unit1.Em4.ControlNodes".sideTapeAttachment."step".transition1[140] )
   END_RUNG
   RUNG wire#w1
      Contact( "Unit1.Em4.ControlNodes".sideTapeAttachment."step".transition1[140] )
      { S7_Templates := "time_type := Time" } #statTonTime[140].TON(pt := T#500ms, et =>)
      wire#w2
      Contact( #unitStatus.specialFunctions."sideTapeRight1 Unuse" )
      Contact( #unitStatus.specialFunctions."sideTapeRight2 Unuse" )
      Contact( #unitStatus.specialFunctions."sideTapeRight3 Unuse" )
      Contact( #unitStatus.specialFunctions."sideTapeRight4 Unuse" )
      Contact( "Unit1.Em4.ControlNodes".cmSideTapeAttachment2TopVaccumOffOn.monitoring.inWorkPos )
      Contact( "Unit1.Em4.ControlNodes".cmSideTapeAttachment2BtmVaccumOffOn.monitoring.inWorkPos )
      Move(in := #JOB_1_STEP_41, out1 => "Unit1.Em4.ControlNodes".sideTapeAttachment.sequence.status.nextStep)
   END_RUNG
   RUNG wire#w2
      I_Contact( "Unit1.Em4.ControlNodes".cmSideTapeAttachment2TopVaccumOffOn.monitoring.inHomePos )
      I_Contact( "Unit1.Em4.ControlNodes".cmSideTapeAttachment2BtmVaccumOffOn.monitoring.inHomePos )
      I_Contact( "Unit1.Em4.ControlNodes".cmSideTapeAttachment2TopVaccumOffOn.monitoring.inWorkPos )
      I_Contact( "Unit1.Em4.ControlNodes".cmSideTapeAttachment2BtmVaccumOffOn.monitoring.inWorkPos )
      Move(in := #JOB_1_STEP_43, out1 => "Unit1.Em4.ControlNodes".sideTapeAttachment.sequence.status.nextStep)
   END_RUNG
   RUNG wire#w2
      I_Contact( #unitStatus.specialFunctions."sideTapeRight1 Unuse" )
      wire#w3
      Move(in := #JOB_1_STEP_80, out1 => "Unit1.Em4.ControlNodes".sideTapeAttachment.sequence.status.nextStep)
   END_RUNG
   RUNG wire#w2
      I_Contact( #unitStatus.specialFunctions."sideTapeRight2 Unuse" )
   END_RUNG wire#w3
   RUNG wire#w2
      I_Contact( #unitStatus.specialFunctions."sideTapeRight3 Unuse" )
   END_RUNG wire#w3
   RUNG wire#w2
      I_Contact( #unitStatus.specialFunctions."sideTapeRight4 Unuse" )
   END_RUNG wire#w3
   RUNG wire#w2
      I_Contact( "Unit1.Em4.ControlNodes".cmSideTapeAttachment2TopVaccumOffOn.monitoring.inWorkPos )
      I_Contact( "Unit1.Em4.ControlNodes".cmSideTapeAttachment2BtmVaccumOffOn.monitoring.inWorkPos )
   END_RUNG wire#w3
   // the same network as SCL:
   "Unit1.Em4.ControlNodes".sideTapeAttachment."step".action1[140] := ("Unit1.Em4.ControlNodes".sideTapeAttachment.sequence.status.currentStep = #JOB_1_STEP_40) AND "Unit1.Em4.ControlNodes".sideTapeAttachment.sequence.status.seqActive;
   "Unit1.Em4.ControlNodes".sideTapeAttachment."step".transition1[140] := ("Unit1.Em4.ControlNodes".sideTapeAttachment.sequence.status.currentStep = #JOB_1_STEP_40) AND "Unit1.Em4.ControlNodes".sideTapeAttachment.sequence.status.seqActive;
   #statTonTime[140].TON(IN := ("Unit1.Em4.ControlNodes".sideTapeAttachment.sequence.status.currentStep = #JOB_1_STEP_40) AND "Unit1.Em4.ControlNodes".sideTapeAttachment.sequence.status.seqActive AND "Unit1.Em4.ControlNodes".sideTapeAttachment."step".transition1[140],
                         PT := T#500ms);
   IF #statTonTime[140].Q AND #unitStatus.specialFunctions."sideTapeRight1 Unuse" AND #unitStatus.specialFunctions."sideTapeRight2 Unuse" AND #unitStatus.specialFunctions."sideTapeRight3 Unuse" AND #unitStatus.specialFunctions."sideTapeRight4 Unuse" AND "Unit1.Em4.ControlNodes".cmSideTapeAttachment2TopVaccumOffOn.monitoring.inWorkPos AND "Unit1.Em4.ControlNodes".cmSideTapeAttachment2BtmVaccumOffOn.monitoring.inWorkPos THEN
       "Unit1.Em4.ControlNodes".sideTapeAttachment.sequence.status.nextStep := #JOB_1_STEP_41;
   END_IF;
   IF #statTonTime[140].Q AND NOT "Unit1.Em4.ControlNodes".cmSideTapeAttachment2TopVaccumOffOn.monitoring.inHomePos AND NOT "Unit1.Em4.ControlNodes".cmSideTapeAttachment2BtmVaccumOffOn.monitoring.inHomePos AND NOT "Unit1.Em4.ControlNodes".cmSideTapeAttachment2TopVaccumOffOn.monitoring.inWorkPos AND NOT "Unit1.Em4.ControlNodes".cmSideTapeAttachment2BtmVaccumOffOn.monitoring.inWorkPos THEN
       "Unit1.Em4.ControlNodes".sideTapeAttachment.sequence.status.nextStep := #JOB_1_STEP_43;
   END_IF;
   IF #statTonTime[140].Q AND (NOT #unitStatus.specialFunctions."sideTapeRight1 Unuse" OR NOT #unitStatus.specialFunctions."sideTapeRight2 Unuse" OR NOT #unitStatus.specialFunctions."sideTapeRight3 Unuse" OR NOT #unitStatus.specialFunctions."sideTapeRight4 Unuse" OR (NOT "Unit1.Em4.ControlNodes".cmSideTapeAttachment2TopVaccumOffOn.monitoring.inWorkPos AND NOT "Unit1.Em4.ControlNodes".cmSideTapeAttachment2BtmVaccumOffOn.monitoring.inWorkPos)) THEN
       "Unit1.Em4.ControlNodes".sideTapeAttachment.sequence.status.nextStep := #JOB_1_STEP_80;
   END_IF;
END_REGION

REGION Network 19: Step[141] : Side Tape Attachment X-Axis Remain Attach Right Position
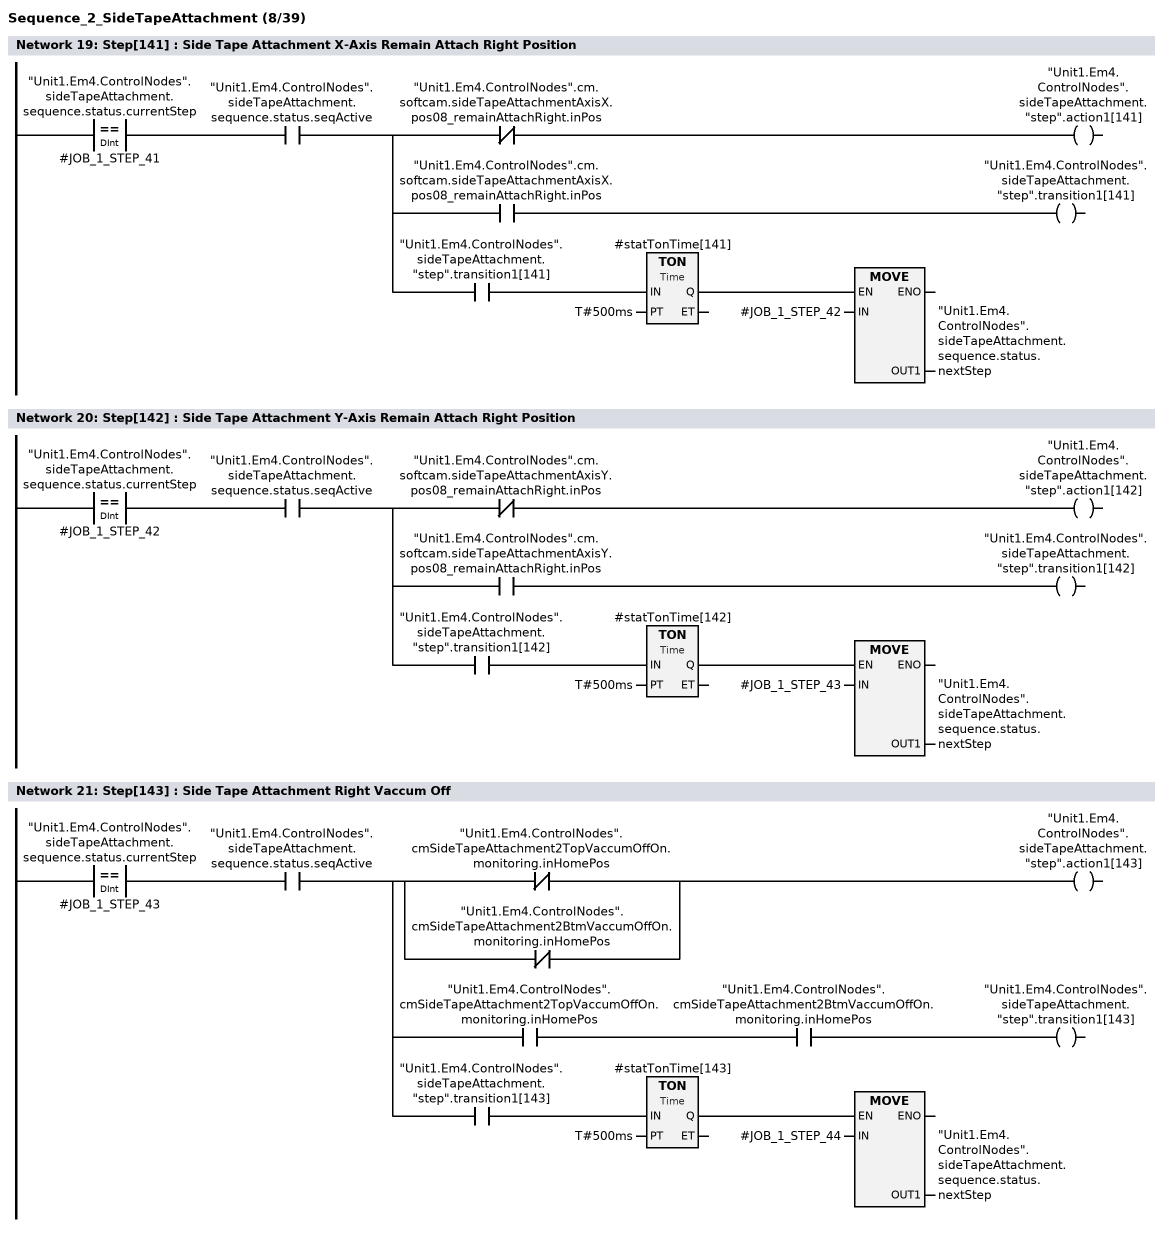
   RUNG wire#powerrail
      { S7_Templates := "SrcType := DInt" } EQ_Contact(in1 := "Unit1.Em4.ControlNodes".sideTapeAttachment.sequence.status.currentStep, in2 := #JOB_1_STEP_41)
      Contact( "Unit1.Em4.ControlNodes".sideTapeAttachment.sequence.status.seqActive )
      wire#w1
      I_Contact( "Unit1.Em4.ControlNodes".cm.softcam.sideTapeAttachmentAxisX.pos08_remainAttachRight.inPos )
      Coil( "Unit1.Em4.ControlNodes".sideTapeAttachment."step".action1[141] )
   END_RUNG
   RUNG wire#w1
      Contact( "Unit1.Em4.ControlNodes".cm.softcam.sideTapeAttachmentAxisX.pos08_remainAttachRight.inPos )
      Coil( "Unit1.Em4.ControlNodes".sideTapeAttachment."step".transition1[141] )
   END_RUNG
   RUNG wire#w1
      Contact( "Unit1.Em4.ControlNodes".sideTapeAttachment."step".transition1[141] )
      { S7_Templates := "time_type := Time" } #statTonTime[141].TON(pt := T#500ms, et =>)
      Move(in := #JOB_1_STEP_42, out1 => "Unit1.Em4.ControlNodes".sideTapeAttachment.sequence.status.nextStep)
   END_RUNG
   // the same network as SCL:
   #_w1 := ("Unit1.Em4.ControlNodes".sideTapeAttachment.sequence.status.currentStep = #JOB_1_STEP_41) AND "Unit1.Em4.ControlNodes".sideTapeAttachment.sequence.status.seqActive;
   "Unit1.Em4.ControlNodes".sideTapeAttachment."step".action1[141] := #_w1 AND NOT "Unit1.Em4.ControlNodes".cm.softcam.sideTapeAttachmentAxisX.pos08_remainAttachRight.inPos;
   "Unit1.Em4.ControlNodes".sideTapeAttachment."step".transition1[141] := #_w1 AND "Unit1.Em4.ControlNodes".cm.softcam.sideTapeAttachmentAxisX.pos08_remainAttachRight.inPos;
   #statTonTime[141].TON(IN := #_w1 AND "Unit1.Em4.ControlNodes".sideTapeAttachment."step".transition1[141],
                         PT := T#500ms);
   IF #statTonTime[141].Q THEN
       "Unit1.Em4.ControlNodes".sideTapeAttachment.sequence.status.nextStep := #JOB_1_STEP_42;
   END_IF;
END_REGION

REGION Network 20: Step[142] : Side Tape Attachment Y-Axis Remain Attach Right Position
   RUNG wire#powerrail
      { S7_Templates := "SrcType := DInt" } EQ_Contact(in1 := "Unit1.Em4.ControlNodes".sideTapeAttachment.sequence.status.currentStep, in2 := #JOB_1_STEP_42)
      Contact( "Unit1.Em4.ControlNodes".sideTapeAttachment.sequence.status.seqActive )
      wire#w1
      I_Contact( "Unit1.Em4.ControlNodes".cm.softcam.sideTapeAttachmentAxisY.pos08_remainAttachRight.inPos )
      Coil( "Unit1.Em4.ControlNodes".sideTapeAttachment."step".action1[142] )
   END_RUNG
   RUNG wire#w1
      Contact( "Unit1.Em4.ControlNodes".cm.softcam.sideTapeAttachmentAxisY.pos08_remainAttachRight.inPos )
      Coil( "Unit1.Em4.ControlNodes".sideTapeAttachment."step".transition1[142] )
   END_RUNG
   RUNG wire#w1
      Contact( "Unit1.Em4.ControlNodes".sideTapeAttachment."step".transition1[142] )
      { S7_Templates := "time_type := Time" } #statTonTime[142].TON(pt := T#500ms, et =>)
      Move(in := #JOB_1_STEP_43, out1 => "Unit1.Em4.ControlNodes".sideTapeAttachment.sequence.status.nextStep)
   END_RUNG
   // the same network as SCL:
   #_w1 := ("Unit1.Em4.ControlNodes".sideTapeAttachment.sequence.status.currentStep = #JOB_1_STEP_42) AND "Unit1.Em4.ControlNodes".sideTapeAttachment.sequence.status.seqActive;
   "Unit1.Em4.ControlNodes".sideTapeAttachment."step".action1[142] := #_w1 AND NOT "Unit1.Em4.ControlNodes".cm.softcam.sideTapeAttachmentAxisY.pos08_remainAttachRight.inPos;
   "Unit1.Em4.ControlNodes".sideTapeAttachment."step".transition1[142] := #_w1 AND "Unit1.Em4.ControlNodes".cm.softcam.sideTapeAttachmentAxisY.pos08_remainAttachRight.inPos;
   #statTonTime[142].TON(IN := #_w1 AND "Unit1.Em4.ControlNodes".sideTapeAttachment."step".transition1[142],
                         PT := T#500ms);
   IF #statTonTime[142].Q THEN
       "Unit1.Em4.ControlNodes".sideTapeAttachment.sequence.status.nextStep := #JOB_1_STEP_43;
   END_IF;
END_REGION

REGION Network 21: Step[143] : Side Tape Attachment Right Vaccum Off
   RUNG wire#powerrail
      { S7_Templates := "SrcType := DInt" } EQ_Contact(in1 := "Unit1.Em4.ControlNodes".sideTapeAttachment.sequence.status.currentStep, in2 := #JOB_1_STEP_43)
      Contact( "Unit1.Em4.ControlNodes".sideTapeAttachment.sequence.status.seqActive )
      wire#w1
      I_Contact( "Unit1.Em4.ControlNodes".cmSideTapeAttachment2TopVaccumOffOn.monitoring.inHomePos )
      wire#w2
      Coil( "Unit1.Em4.ControlNodes".sideTapeAttachment."step".action1[143] )
   END_RUNG
   RUNG wire#w1
      I_Contact( "Unit1.Em4.ControlNodes".cmSideTapeAttachment2BtmVaccumOffOn.monitoring.inHomePos )
   END_RUNG wire#w2
   RUNG wire#w1
      Contact( "Unit1.Em4.ControlNodes".cmSideTapeAttachment2TopVaccumOffOn.monitoring.inHomePos )
      Contact( "Unit1.Em4.ControlNodes".cmSideTapeAttachment2BtmVaccumOffOn.monitoring.inHomePos )
      Coil( "Unit1.Em4.ControlNodes".sideTapeAttachment."step".transition1[143] )
   END_RUNG
   RUNG wire#w1
      Contact( "Unit1.Em4.ControlNodes".sideTapeAttachment."step".transition1[143] )
      { S7_Templates := "time_type := Time" } #statTonTime[143].TON(pt := T#500ms, et =>)
      Move(in := #JOB_1_STEP_44, out1 => "Unit1.Em4.ControlNodes".sideTapeAttachment.sequence.status.nextStep)
   END_RUNG
   // the same network as SCL:
   #_w1 := ("Unit1.Em4.ControlNodes".sideTapeAttachment.sequence.status.currentStep = #JOB_1_STEP_43) AND "Unit1.Em4.ControlNodes".sideTapeAttachment.sequence.status.seqActive;
   "Unit1.Em4.ControlNodes".sideTapeAttachment."step".action1[143] := #_w1 AND (NOT "Unit1.Em4.ControlNodes".cmSideTapeAttachment2TopVaccumOffOn.monitoring.inHomePos OR NOT "Unit1.Em4.ControlNodes".cmSideTapeAttachment2BtmVaccumOffOn.monitoring.inHomePos);
   "Unit1.Em4.ControlNodes".sideTapeAttachment."step".transition1[143] := #_w1 AND "Unit1.Em4.ControlNodes".cmSideTapeAttachment2TopVaccumOffOn.monitoring.inHomePos AND "Unit1.Em4.ControlNodes".cmSideTapeAttachment2BtmVaccumOffOn.monitoring.inHomePos;
   #statTonTime[143].TON(IN := #_w1 AND "Unit1.Em4.ControlNodes".sideTapeAttachment."step".transition1[143],
                         PT := T#500ms);
   IF #statTonTime[143].Q THEN
       "Unit1.Em4.ControlNodes".sideTapeAttachment.sequence.status.nextStep := #JOB_1_STEP_44;
   END_IF;
END_REGION

REGION Network 22: Step[144] : Side Tape Attachment Y-Axis Wait Pos
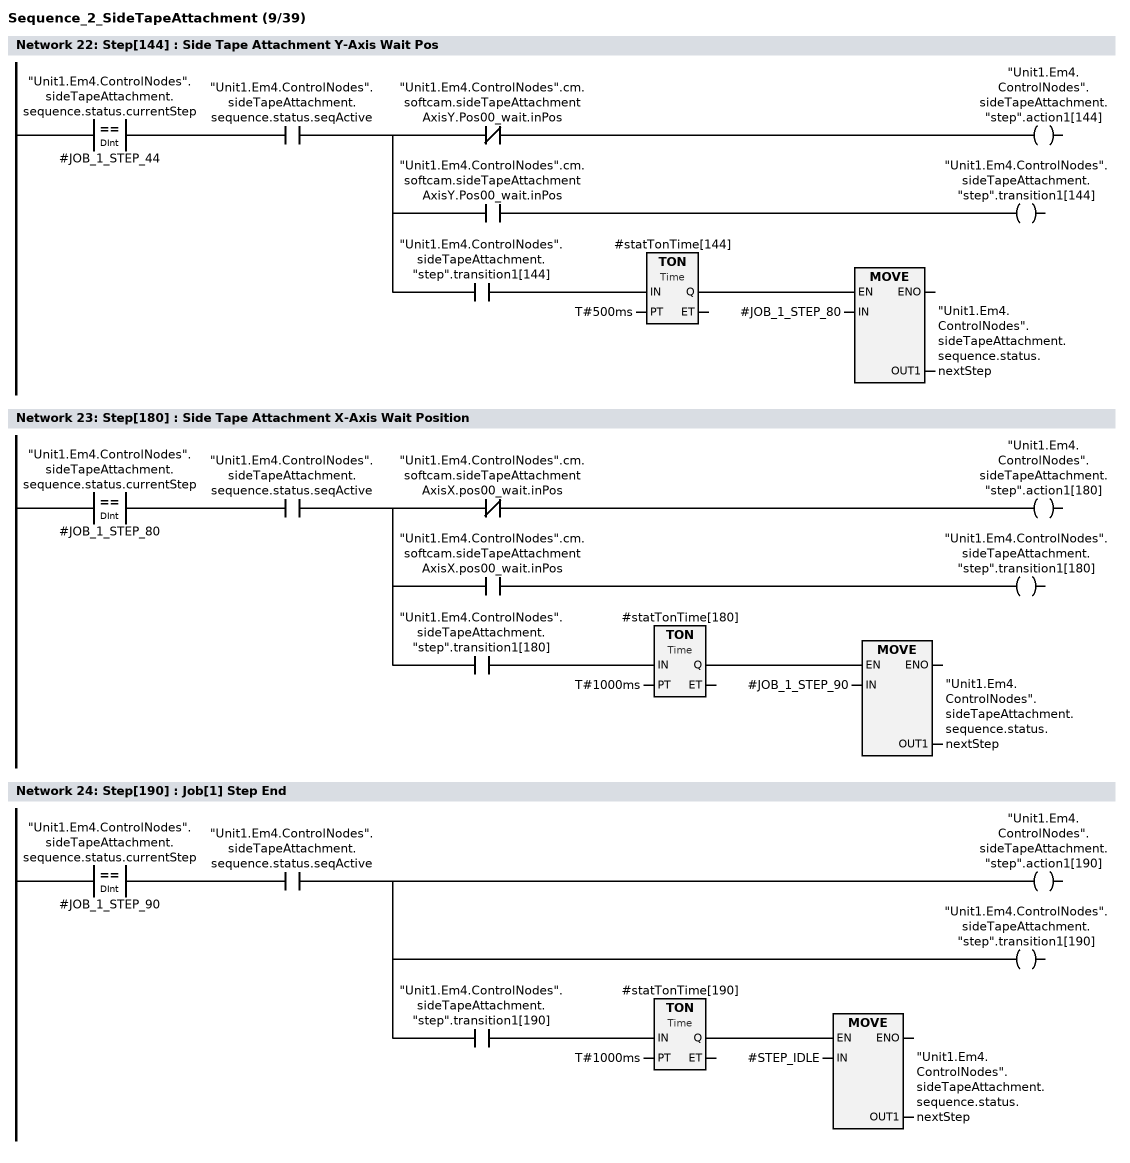
   RUNG wire#powerrail
      { S7_Templates := "SrcType := DInt" } EQ_Contact(in1 := "Unit1.Em4.ControlNodes".sideTapeAttachment.sequence.status.currentStep, in2 := #JOB_1_STEP_44)
      Contact( "Unit1.Em4.ControlNodes".sideTapeAttachment.sequence.status.seqActive )
      wire#w1
      I_Contact( "Unit1.Em4.ControlNodes".cm.softcam.sideTapeAttachmentAxisY.Pos00_wait.inPos )
      Coil( "Unit1.Em4.ControlNodes".sideTapeAttachment."step".action1[144] )
   END_RUNG
   RUNG wire#w1
      Contact( "Unit1.Em4.ControlNodes".cm.softcam.sideTapeAttachmentAxisY.Pos00_wait.inPos )
      Coil( "Unit1.Em4.ControlNodes".sideTapeAttachment."step".transition1[144] )
   END_RUNG
   RUNG wire#w1
      Contact( "Unit1.Em4.ControlNodes".sideTapeAttachment."step".transition1[144] )
      { S7_Templates := "time_type := Time" } #statTonTime[144].TON(pt := T#500ms, et =>)
      Move(in := #JOB_1_STEP_80, out1 => "Unit1.Em4.ControlNodes".sideTapeAttachment.sequence.status.nextStep)
   END_RUNG
   // the same network as SCL:
   #_w1 := ("Unit1.Em4.ControlNodes".sideTapeAttachment.sequence.status.currentStep = #JOB_1_STEP_44) AND "Unit1.Em4.ControlNodes".sideTapeAttachment.sequence.status.seqActive;
   "Unit1.Em4.ControlNodes".sideTapeAttachment."step".action1[144] := #_w1 AND NOT "Unit1.Em4.ControlNodes".cm.softcam.sideTapeAttachmentAxisY.Pos00_wait.inPos;
   "Unit1.Em4.ControlNodes".sideTapeAttachment."step".transition1[144] := #_w1 AND "Unit1.Em4.ControlNodes".cm.softcam.sideTapeAttachmentAxisY.Pos00_wait.inPos;
   #statTonTime[144].TON(IN := #_w1 AND "Unit1.Em4.ControlNodes".sideTapeAttachment."step".transition1[144],
                         PT := T#500ms);
   IF #statTonTime[144].Q THEN
       "Unit1.Em4.ControlNodes".sideTapeAttachment.sequence.status.nextStep := #JOB_1_STEP_80;
   END_IF;
END_REGION

REGION Network 23: Step[180] : Side Tape Attachment X-Axis Wait Position
   RUNG wire#powerrail
      { S7_Templates := "SrcType := DInt" } EQ_Contact(in1 := "Unit1.Em4.ControlNodes".sideTapeAttachment.sequence.status.currentStep, in2 := #JOB_1_STEP_80)
      Contact( "Unit1.Em4.ControlNodes".sideTapeAttachment.sequence.status.seqActive )
      wire#w1
      I_Contact( "Unit1.Em4.ControlNodes".cm.softcam.sideTapeAttachmentAxisX.pos00_wait.inPos )
      Coil( "Unit1.Em4.ControlNodes".sideTapeAttachment."step".action1[180] )
   END_RUNG
   RUNG wire#w1
      Contact( "Unit1.Em4.ControlNodes".cm.softcam.sideTapeAttachmentAxisX.pos00_wait.inPos )
      Coil( "Unit1.Em4.ControlNodes".sideTapeAttachment."step".transition1[180] )
   END_RUNG
   RUNG wire#w1
      Contact( "Unit1.Em4.ControlNodes".sideTapeAttachment."step".transition1[180] )
      { S7_Templates := "time_type := Time" } #statTonTime[180].TON(pt := T#1000ms, et =>)
      Move(in := #JOB_1_STEP_90, out1 => "Unit1.Em4.ControlNodes".sideTapeAttachment.sequence.status.nextStep)
   END_RUNG
   // the same network as SCL:
   #_w1 := ("Unit1.Em4.ControlNodes".sideTapeAttachment.sequence.status.currentStep = #JOB_1_STEP_80) AND "Unit1.Em4.ControlNodes".sideTapeAttachment.sequence.status.seqActive;
   "Unit1.Em4.ControlNodes".sideTapeAttachment."step".action1[180] := #_w1 AND NOT "Unit1.Em4.ControlNodes".cm.softcam.sideTapeAttachmentAxisX.pos00_wait.inPos;
   "Unit1.Em4.ControlNodes".sideTapeAttachment."step".transition1[180] := #_w1 AND "Unit1.Em4.ControlNodes".cm.softcam.sideTapeAttachmentAxisX.pos00_wait.inPos;
   #statTonTime[180].TON(IN := #_w1 AND "Unit1.Em4.ControlNodes".sideTapeAttachment."step".transition1[180],
                         PT := T#1000ms);
   IF #statTonTime[180].Q THEN
       "Unit1.Em4.ControlNodes".sideTapeAttachment.sequence.status.nextStep := #JOB_1_STEP_90;
   END_IF;
END_REGION

REGION Network 24: Step[190] : Job[1] Step End
   RUNG wire#powerrail
      { S7_Templates := "SrcType := DInt" } EQ_Contact(in1 := "Unit1.Em4.ControlNodes".sideTapeAttachment.sequence.status.currentStep, in2 := #JOB_1_STEP_90)
      Contact( "Unit1.Em4.ControlNodes".sideTapeAttachment.sequence.status.seqActive )
      wire#w1
      Coil( "Unit1.Em4.ControlNodes".sideTapeAttachment."step".action1[190] )
   END_RUNG
   RUNG wire#w1
      Coil( "Unit1.Em4.ControlNodes".sideTapeAttachment."step".transition1[190] )
   END_RUNG
   RUNG wire#w1
      Contact( "Unit1.Em4.ControlNodes".sideTapeAttachment."step".transition1[190] )
      { S7_Templates := "time_type := Time" } #statTonTime[190].TON(pt := T#1000ms, et =>)
      Move(in := #STEP_IDLE, out1 => "Unit1.Em4.ControlNodes".sideTapeAttachment.sequence.status.nextStep)
   END_RUNG
   // the same network as SCL:
   "Unit1.Em4.ControlNodes".sideTapeAttachment."step".action1[190] := ("Unit1.Em4.ControlNodes".sideTapeAttachment.sequence.status.currentStep = #JOB_1_STEP_90) AND "Unit1.Em4.ControlNodes".sideTapeAttachment.sequence.status.seqActive;
   "Unit1.Em4.ControlNodes".sideTapeAttachment."step".transition1[190] := ("Unit1.Em4.ControlNodes".sideTapeAttachment.sequence.status.currentStep = #JOB_1_STEP_90) AND "Unit1.Em4.ControlNodes".sideTapeAttachment.sequence.status.seqActive;
   #statTonTime[190].TON(IN := ("Unit1.Em4.ControlNodes".sideTapeAttachment.sequence.status.currentStep = #JOB_1_STEP_90) AND "Unit1.Em4.ControlNodes".sideTapeAttachment.sequence.status.seqActive AND "Unit1.Em4.ControlNodes".sideTapeAttachment."step".transition1[190],
                         PT := T#1000ms);
   IF #statTonTime[190].Q THEN
       "Unit1.Em4.ControlNodes".sideTapeAttachment.sequence.status.nextStep := #STEP_IDLE;
   END_IF;
END_REGION

REGION Network 25: *************** JOB[2] SIDE TAPE RIGHT GET=AUTO *************************
END_REGION

REGION Network 26: Step[201] : JOB[2] Condition
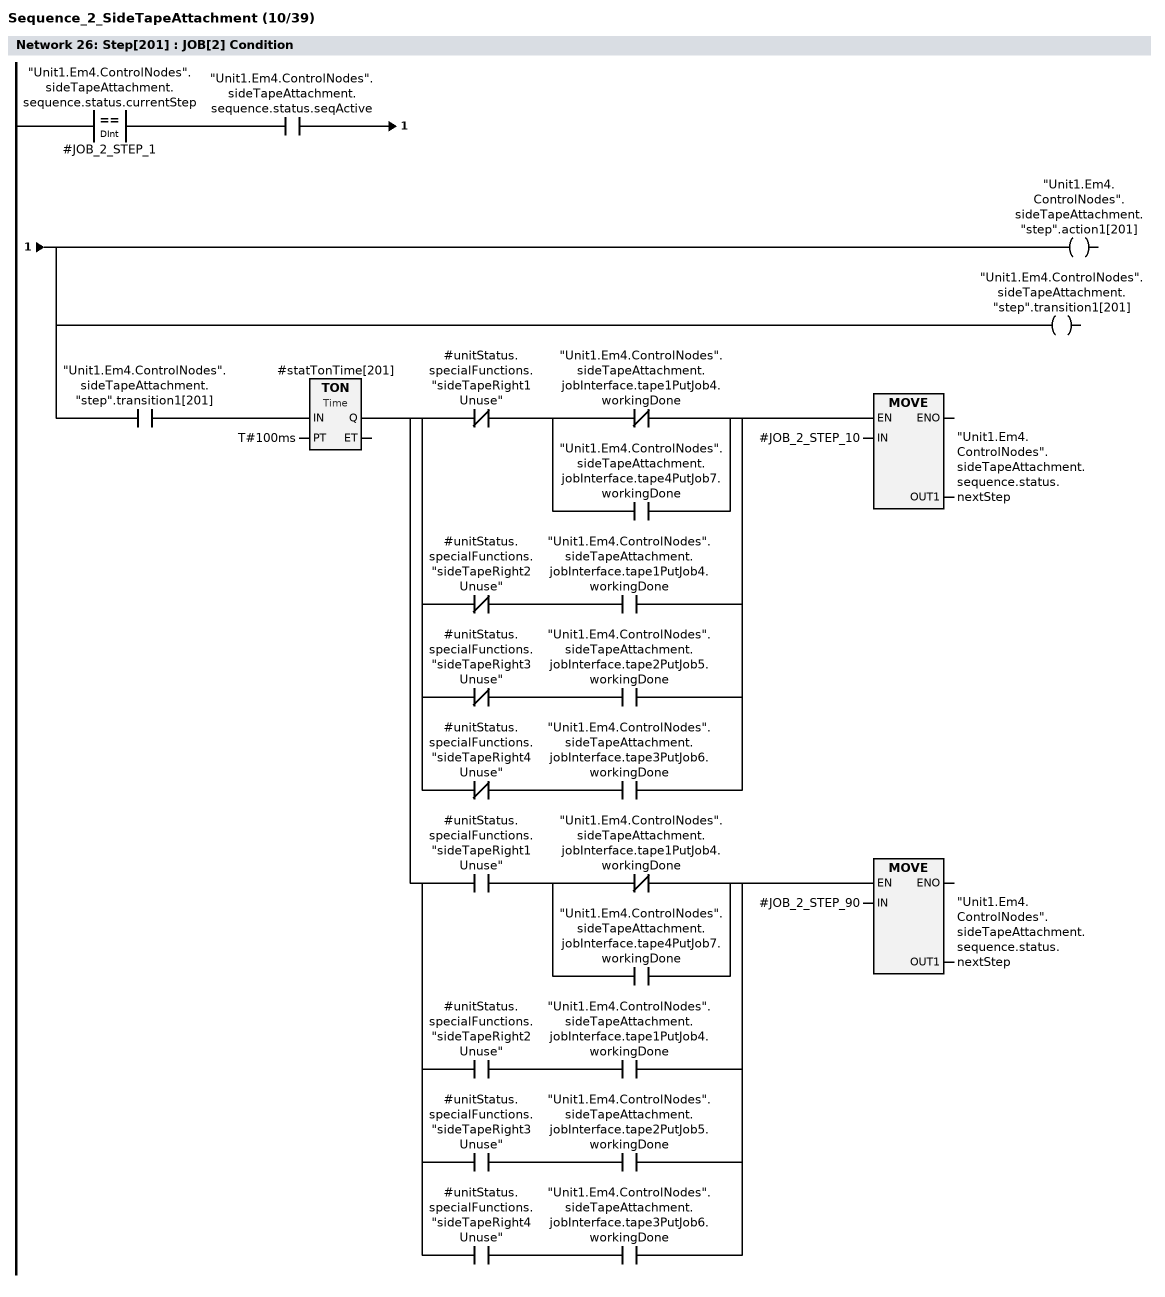
   RUNG wire#powerrail
      { S7_Templates := "SrcType := DInt" } EQ_Contact(in1 := "Unit1.Em4.ControlNodes".sideTapeAttachment.sequence.status.currentStep, in2 := #JOB_2_STEP_1)
      Contact( "Unit1.Em4.ControlNodes".sideTapeAttachment.sequence.status.seqActive )
      wire#w1
      Coil( "Unit1.Em4.ControlNodes".sideTapeAttachment."step".action1[201] )
   END_RUNG
   RUNG wire#w1
      Coil( "Unit1.Em4.ControlNodes".sideTapeAttachment."step".transition1[201] )
   END_RUNG
   RUNG wire#w1
      Contact( "Unit1.Em4.ControlNodes".sideTapeAttachment."step".transition1[201] )
      { S7_Templates := "time_type := Time" } #statTonTime[201].TON(pt := T#100ms, et =>)
      wire#w2
      I_Contact( #unitStatus.specialFunctions."sideTapeRight1 Unuse" )
      wire#w3
      I_Contact( "Unit1.Em4.ControlNodes".sideTapeAttachment.jobInterface.tape1PutJob4.workingDone )
      wire#w4
      Move(in := #JOB_2_STEP_10, out1 => "Unit1.Em4.ControlNodes".sideTapeAttachment.sequence.status.nextStep)
   END_RUNG
   RUNG wire#w3
      Contact( "Unit1.Em4.ControlNodes".sideTapeAttachment.jobInterface.tape4PutJob7.workingDone )
   END_RUNG wire#w4
   RUNG wire#w2
      I_Contact( #unitStatus.specialFunctions."sideTapeRight2 Unuse" )
      Contact( "Unit1.Em4.ControlNodes".sideTapeAttachment.jobInterface.tape1PutJob4.workingDone )
   END_RUNG wire#w4
   RUNG wire#w2
      I_Contact( #unitStatus.specialFunctions."sideTapeRight3 Unuse" )
      Contact( "Unit1.Em4.ControlNodes".sideTapeAttachment.jobInterface.tape2PutJob5.workingDone )
   END_RUNG wire#w4
   RUNG wire#w2
      I_Contact( #unitStatus.specialFunctions."sideTapeRight4 Unuse" )
      Contact( "Unit1.Em4.ControlNodes".sideTapeAttachment.jobInterface.tape3PutJob6.workingDone )
   END_RUNG wire#w4
   RUNG wire#w2
      Contact( #unitStatus.specialFunctions."sideTapeRight1 Unuse" )
      wire#w5
      I_Contact( "Unit1.Em4.ControlNodes".sideTapeAttachment.jobInterface.tape1PutJob4.workingDone )
      wire#w6
      Move(in := #JOB_2_STEP_90, out1 => "Unit1.Em4.ControlNodes".sideTapeAttachment.sequence.status.nextStep)
   END_RUNG
   RUNG wire#w5
      Contact( "Unit1.Em4.ControlNodes".sideTapeAttachment.jobInterface.tape4PutJob7.workingDone )
   END_RUNG wire#w6
   RUNG wire#w2
      Contact( #unitStatus.specialFunctions."sideTapeRight2 Unuse" )
      Contact( "Unit1.Em4.ControlNodes".sideTapeAttachment.jobInterface.tape1PutJob4.workingDone )
   END_RUNG wire#w6
   RUNG wire#w2
      Contact( #unitStatus.specialFunctions."sideTapeRight3 Unuse" )
      Contact( "Unit1.Em4.ControlNodes".sideTapeAttachment.jobInterface.tape2PutJob5.workingDone )
   END_RUNG wire#w6
   RUNG wire#w2
      Contact( #unitStatus.specialFunctions."sideTapeRight4 Unuse" )
      Contact( "Unit1.Em4.ControlNodes".sideTapeAttachment.jobInterface.tape3PutJob6.workingDone )
   END_RUNG wire#w6
   // the same network as SCL:
   "Unit1.Em4.ControlNodes".sideTapeAttachment."step".action1[201] := ("Unit1.Em4.ControlNodes".sideTapeAttachment.sequence.status.currentStep = #JOB_2_STEP_1) AND "Unit1.Em4.ControlNodes".sideTapeAttachment.sequence.status.seqActive;
   "Unit1.Em4.ControlNodes".sideTapeAttachment."step".transition1[201] := ("Unit1.Em4.ControlNodes".sideTapeAttachment.sequence.status.currentStep = #JOB_2_STEP_1) AND "Unit1.Em4.ControlNodes".sideTapeAttachment.sequence.status.seqActive;
   #statTonTime[201].TON(IN := ("Unit1.Em4.ControlNodes".sideTapeAttachment.sequence.status.currentStep = #JOB_2_STEP_1) AND "Unit1.Em4.ControlNodes".sideTapeAttachment.sequence.status.seqActive AND "Unit1.Em4.ControlNodes".sideTapeAttachment."step".transition1[201],
                         PT := T#100ms);
   IF #statTonTime[201].Q AND ((NOT #unitStatus.specialFunctions."sideTapeRight1 Unuse" AND (NOT "Unit1.Em4.ControlNodes".sideTapeAttachment.jobInterface.tape1PutJob4.workingDone OR "Unit1.Em4.ControlNodes".sideTapeAttachment.jobInterface.tape4PutJob7.workingDone)) OR (NOT #unitStatus.specialFunctions."sideTapeRight2 Unuse" AND "Unit1.Em4.ControlNodes".sideTapeAttachment.jobInterface.tape1PutJob4.workingDone) OR (NOT #unitStatus.specialFunctions."sideTapeRight3 Unuse" AND "Unit1.Em4.ControlNodes".sideTapeAttachment.jobInterface.tape2PutJob5.workingDone) OR (NOT #unitStatus.specialFunctions."sideTapeRight4 Unuse" AND "Unit1.Em4.ControlNodes".sideTapeAttachment.jobInterface.tape3PutJob6.workingDone)) THEN
       "Unit1.Em4.ControlNodes".sideTapeAttachment.sequence.status.nextStep := #JOB_2_STEP_10;
   END_IF;
   IF #statTonTime[201].Q AND ((#unitStatus.specialFunctions."sideTapeRight1 Unuse" AND (NOT "Unit1.Em4.ControlNodes".sideTapeAttachment.jobInterface.tape1PutJob4.workingDone OR "Unit1.Em4.ControlNodes".sideTapeAttachment.jobInterface.tape4PutJob7.workingDone)) OR (#unitStatus.specialFunctions."sideTapeRight2 Unuse" AND "Unit1.Em4.ControlNodes".sideTapeAttachment.jobInterface.tape1PutJob4.workingDone) OR (#unitStatus.specialFunctions."sideTapeRight3 Unuse" AND "Unit1.Em4.ControlNodes".sideTapeAttachment.jobInterface.tape2PutJob5.workingDone) OR (#unitStatus.specialFunctions."sideTapeRight4 Unuse" AND "Unit1.Em4.ControlNodes".sideTapeAttachment.jobInterface.tape3PutJob6.workingDone)) THEN
       "Unit1.Em4.ControlNodes".sideTapeAttachment.sequence.status.nextStep := #JOB_2_STEP_90;
   END_IF;
END_REGION

REGION Network 27: Step[210] : Side Tape Attachment X-Axis Right Tape Get Pos
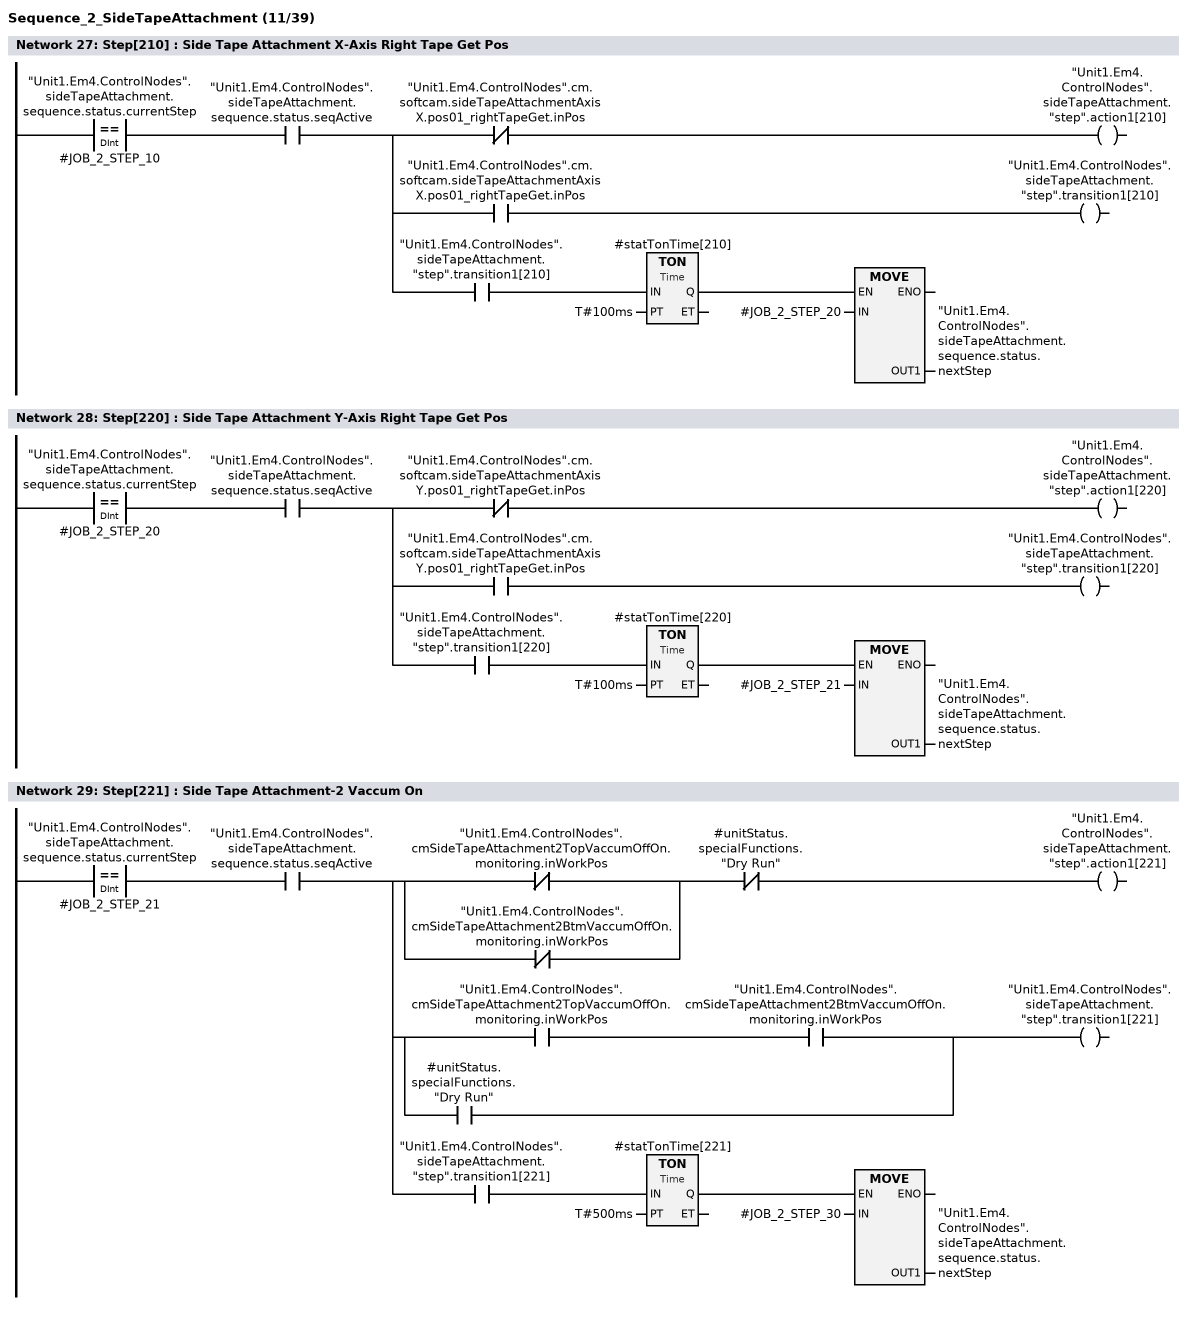
   RUNG wire#powerrail
      { S7_Templates := "SrcType := DInt" } EQ_Contact(in1 := "Unit1.Em4.ControlNodes".sideTapeAttachment.sequence.status.currentStep, in2 := #JOB_2_STEP_10)
      Contact( "Unit1.Em4.ControlNodes".sideTapeAttachment.sequence.status.seqActive )
      wire#w1
      I_Contact( "Unit1.Em4.ControlNodes".cm.softcam.sideTapeAttachmentAxisX.pos01_rightTapeGet.inPos )
      Coil( "Unit1.Em4.ControlNodes".sideTapeAttachment."step".action1[210] )
   END_RUNG
   RUNG wire#w1
      Contact( "Unit1.Em4.ControlNodes".cm.softcam.sideTapeAttachmentAxisX.pos01_rightTapeGet.inPos )
      Coil( "Unit1.Em4.ControlNodes".sideTapeAttachment."step".transition1[210] )
   END_RUNG
   RUNG wire#w1
      Contact( "Unit1.Em4.ControlNodes".sideTapeAttachment."step".transition1[210] )
      { S7_Templates := "time_type := Time" } #statTonTime[210].TON(pt := T#100ms, et =>)
      Move(in := #JOB_2_STEP_20, out1 => "Unit1.Em4.ControlNodes".sideTapeAttachment.sequence.status.nextStep)
   END_RUNG
   // the same network as SCL:
   #_w1 := ("Unit1.Em4.ControlNodes".sideTapeAttachment.sequence.status.currentStep = #JOB_2_STEP_10) AND "Unit1.Em4.ControlNodes".sideTapeAttachment.sequence.status.seqActive;
   "Unit1.Em4.ControlNodes".sideTapeAttachment."step".action1[210] := #_w1 AND NOT "Unit1.Em4.ControlNodes".cm.softcam.sideTapeAttachmentAxisX.pos01_rightTapeGet.inPos;
   "Unit1.Em4.ControlNodes".sideTapeAttachment."step".transition1[210] := #_w1 AND "Unit1.Em4.ControlNodes".cm.softcam.sideTapeAttachmentAxisX.pos01_rightTapeGet.inPos;
   #statTonTime[210].TON(IN := #_w1 AND "Unit1.Em4.ControlNodes".sideTapeAttachment."step".transition1[210],
                         PT := T#100ms);
   IF #statTonTime[210].Q THEN
       "Unit1.Em4.ControlNodes".sideTapeAttachment.sequence.status.nextStep := #JOB_2_STEP_20;
   END_IF;
END_REGION

REGION Network 28: Step[220] : Side Tape Attachment Y-Axis Right Tape Get Pos
   RUNG wire#powerrail
      { S7_Templates := "SrcType := DInt" } EQ_Contact(in1 := "Unit1.Em4.ControlNodes".sideTapeAttachment.sequence.status.currentStep, in2 := #JOB_2_STEP_20)
      Contact( "Unit1.Em4.ControlNodes".sideTapeAttachment.sequence.status.seqActive )
      wire#w1
      I_Contact( "Unit1.Em4.ControlNodes".cm.softcam.sideTapeAttachmentAxisY.pos01_rightTapeGet.inPos )
      Coil( "Unit1.Em4.ControlNodes".sideTapeAttachment."step".action1[220] )
   END_RUNG
   RUNG wire#w1
      Contact( "Unit1.Em4.ControlNodes".cm.softcam.sideTapeAttachmentAxisY.pos01_rightTapeGet.inPos )
      Coil( "Unit1.Em4.ControlNodes".sideTapeAttachment."step".transition1[220] )
   END_RUNG
   RUNG wire#w1
      Contact( "Unit1.Em4.ControlNodes".sideTapeAttachment."step".transition1[220] )
      { S7_Templates := "time_type := Time" } #statTonTime[220].TON(pt := T#100ms, et =>)
      Move(in := #JOB_2_STEP_21, out1 => "Unit1.Em4.ControlNodes".sideTapeAttachment.sequence.status.nextStep)
   END_RUNG
   // the same network as SCL:
   #_w1 := ("Unit1.Em4.ControlNodes".sideTapeAttachment.sequence.status.currentStep = #JOB_2_STEP_20) AND "Unit1.Em4.ControlNodes".sideTapeAttachment.sequence.status.seqActive;
   "Unit1.Em4.ControlNodes".sideTapeAttachment."step".action1[220] := #_w1 AND NOT "Unit1.Em4.ControlNodes".cm.softcam.sideTapeAttachmentAxisY.pos01_rightTapeGet.inPos;
   "Unit1.Em4.ControlNodes".sideTapeAttachment."step".transition1[220] := #_w1 AND "Unit1.Em4.ControlNodes".cm.softcam.sideTapeAttachmentAxisY.pos01_rightTapeGet.inPos;
   #statTonTime[220].TON(IN := #_w1 AND "Unit1.Em4.ControlNodes".sideTapeAttachment."step".transition1[220],
                         PT := T#100ms);
   IF #statTonTime[220].Q THEN
       "Unit1.Em4.ControlNodes".sideTapeAttachment.sequence.status.nextStep := #JOB_2_STEP_21;
   END_IF;
END_REGION

REGION Network 29: Step[221] : Side Tape Attachment-2 Vaccum On
   RUNG wire#powerrail
      { S7_Templates := "SrcType := DInt" } EQ_Contact(in1 := "Unit1.Em4.ControlNodes".sideTapeAttachment.sequence.status.currentStep, in2 := #JOB_2_STEP_21)
      Contact( "Unit1.Em4.ControlNodes".sideTapeAttachment.sequence.status.seqActive )
      wire#w1
      I_Contact( "Unit1.Em4.ControlNodes".cmSideTapeAttachment2TopVaccumOffOn.monitoring.inWorkPos )
      wire#w2
      I_Contact( #unitStatus.specialFunctions."Dry Run" )
      Coil( "Unit1.Em4.ControlNodes".sideTapeAttachment."step".action1[221] )
   END_RUNG
   RUNG wire#w1
      I_Contact( "Unit1.Em4.ControlNodes".cmSideTapeAttachment2BtmVaccumOffOn.monitoring.inWorkPos )
   END_RUNG wire#w2
   RUNG wire#w1
      Contact( "Unit1.Em4.ControlNodes".cmSideTapeAttachment2TopVaccumOffOn.monitoring.inWorkPos )
      Contact( "Unit1.Em4.ControlNodes".cmSideTapeAttachment2BtmVaccumOffOn.monitoring.inWorkPos )
      wire#w3
      Coil( "Unit1.Em4.ControlNodes".sideTapeAttachment."step".transition1[221] )
   END_RUNG
   RUNG wire#w1
      Contact( #unitStatus.specialFunctions."Dry Run" )
   END_RUNG wire#w3
   RUNG wire#w1
      Contact( "Unit1.Em4.ControlNodes".sideTapeAttachment."step".transition1[221] )
      { S7_Templates := "time_type := Time" } #statTonTime[221].TON(pt := T#500ms, et =>)
      Move(in := #JOB_2_STEP_30, out1 => "Unit1.Em4.ControlNodes".sideTapeAttachment.sequence.status.nextStep)
   END_RUNG
   // the same network as SCL:
   #_w1 := ("Unit1.Em4.ControlNodes".sideTapeAttachment.sequence.status.currentStep = #JOB_2_STEP_21) AND "Unit1.Em4.ControlNodes".sideTapeAttachment.sequence.status.seqActive;
   "Unit1.Em4.ControlNodes".sideTapeAttachment."step".action1[221] := #_w1 AND (NOT "Unit1.Em4.ControlNodes".cmSideTapeAttachment2TopVaccumOffOn.monitoring.inWorkPos OR NOT "Unit1.Em4.ControlNodes".cmSideTapeAttachment2BtmVaccumOffOn.monitoring.inWorkPos) AND NOT #unitStatus.specialFunctions."Dry Run";
   "Unit1.Em4.ControlNodes".sideTapeAttachment."step".transition1[221] := #_w1 AND (("Unit1.Em4.ControlNodes".cmSideTapeAttachment2TopVaccumOffOn.monitoring.inWorkPos AND "Unit1.Em4.ControlNodes".cmSideTapeAttachment2BtmVaccumOffOn.monitoring.inWorkPos) OR #unitStatus.specialFunctions."Dry Run");
   #statTonTime[221].TON(IN := #_w1 AND "Unit1.Em4.ControlNodes".sideTapeAttachment."step".transition1[221],
                         PT := T#500ms);
   IF #statTonTime[221].Q THEN
       "Unit1.Em4.ControlNodes".sideTapeAttachment.sequence.status.nextStep := #JOB_2_STEP_30;
   END_IF;
END_REGION

REGION Network 30: Step[230] : Side Tape Cutter Forward
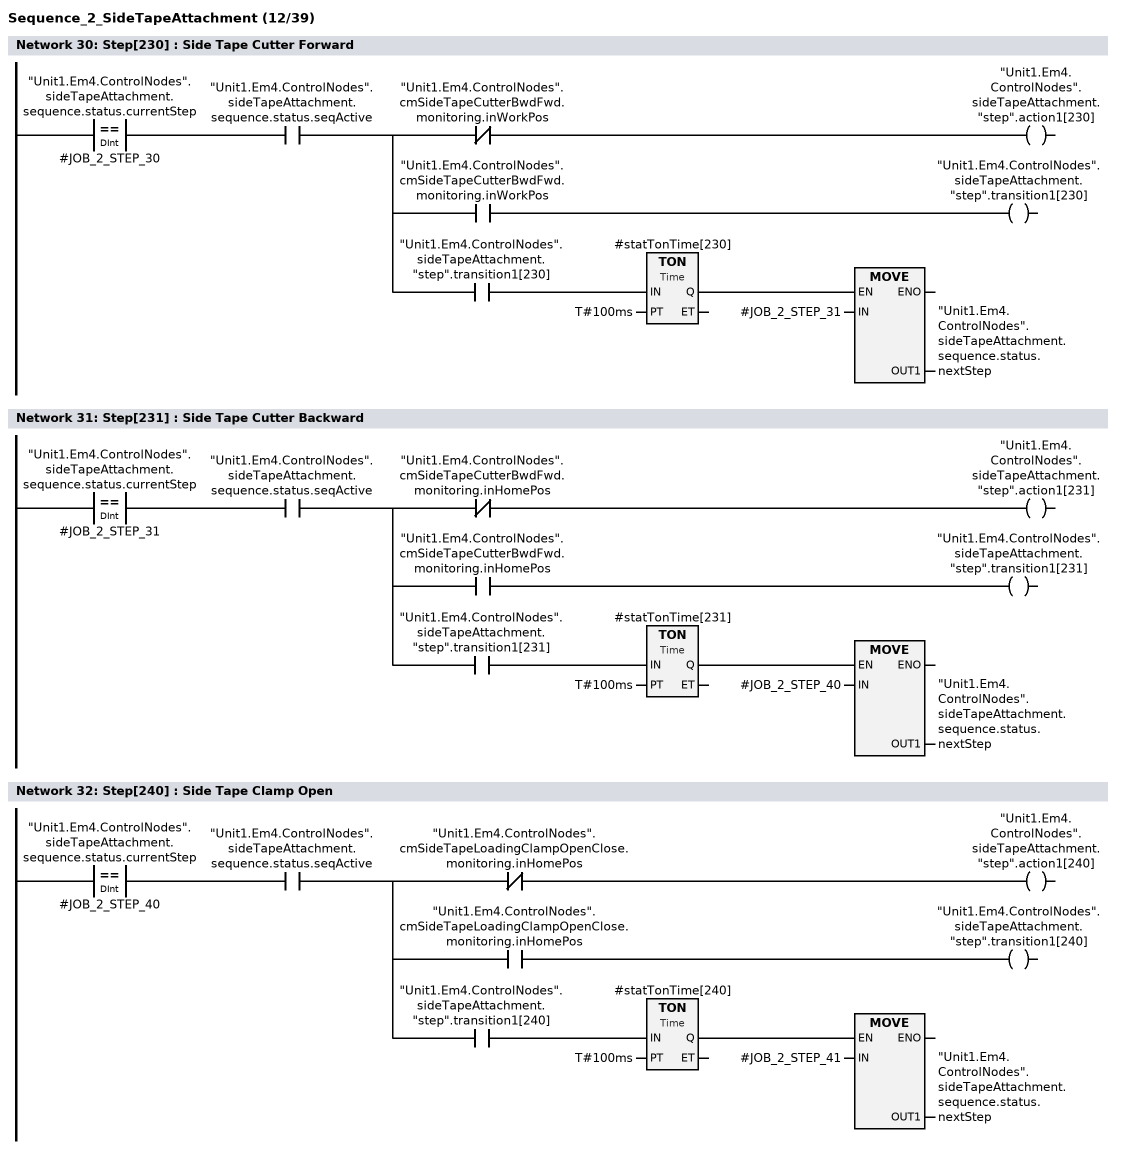
   RUNG wire#powerrail
      { S7_Templates := "SrcType := DInt" } EQ_Contact(in1 := "Unit1.Em4.ControlNodes".sideTapeAttachment.sequence.status.currentStep, in2 := #JOB_2_STEP_30)
      Contact( "Unit1.Em4.ControlNodes".sideTapeAttachment.sequence.status.seqActive )
      wire#w1
      I_Contact( "Unit1.Em4.ControlNodes".cmSideTapeCutterBwdFwd.monitoring.inWorkPos )
      Coil( "Unit1.Em4.ControlNodes".sideTapeAttachment."step".action1[230] )
   END_RUNG
   RUNG wire#w1
      Contact( "Unit1.Em4.ControlNodes".cmSideTapeCutterBwdFwd.monitoring.inWorkPos )
      Coil( "Unit1.Em4.ControlNodes".sideTapeAttachment."step".transition1[230] )
   END_RUNG
   RUNG wire#w1
      Contact( "Unit1.Em4.ControlNodes".sideTapeAttachment."step".transition1[230] )
      { S7_Templates := "time_type := Time" } #statTonTime[230].TON(pt := T#100ms, et =>)
      Move(in := #JOB_2_STEP_31, out1 => "Unit1.Em4.ControlNodes".sideTapeAttachment.sequence.status.nextStep)
   END_RUNG
   // the same network as SCL:
   #_w1 := ("Unit1.Em4.ControlNodes".sideTapeAttachment.sequence.status.currentStep = #JOB_2_STEP_30) AND "Unit1.Em4.ControlNodes".sideTapeAttachment.sequence.status.seqActive;
   "Unit1.Em4.ControlNodes".sideTapeAttachment."step".action1[230] := #_w1 AND NOT "Unit1.Em4.ControlNodes".cmSideTapeCutterBwdFwd.monitoring.inWorkPos;
   "Unit1.Em4.ControlNodes".sideTapeAttachment."step".transition1[230] := #_w1 AND "Unit1.Em4.ControlNodes".cmSideTapeCutterBwdFwd.monitoring.inWorkPos;
   #statTonTime[230].TON(IN := #_w1 AND "Unit1.Em4.ControlNodes".sideTapeAttachment."step".transition1[230],
                         PT := T#100ms);
   IF #statTonTime[230].Q THEN
       "Unit1.Em4.ControlNodes".sideTapeAttachment.sequence.status.nextStep := #JOB_2_STEP_31;
   END_IF;
END_REGION

REGION Network 31: Step[231] : Side Tape Cutter Backward
   RUNG wire#powerrail
      { S7_Templates := "SrcType := DInt" } EQ_Contact(in1 := "Unit1.Em4.ControlNodes".sideTapeAttachment.sequence.status.currentStep, in2 := #JOB_2_STEP_31)
      Contact( "Unit1.Em4.ControlNodes".sideTapeAttachment.sequence.status.seqActive )
      wire#w1
      I_Contact( "Unit1.Em4.ControlNodes".cmSideTapeCutterBwdFwd.monitoring.inHomePos )
      Coil( "Unit1.Em4.ControlNodes".sideTapeAttachment."step".action1[231] )
   END_RUNG
   RUNG wire#w1
      Contact( "Unit1.Em4.ControlNodes".cmSideTapeCutterBwdFwd.monitoring.inHomePos )
      Coil( "Unit1.Em4.ControlNodes".sideTapeAttachment."step".transition1[231] )
   END_RUNG
   RUNG wire#w1
      Contact( "Unit1.Em4.ControlNodes".sideTapeAttachment."step".transition1[231] )
      { S7_Templates := "time_type := Time" } #statTonTime[231].TON(pt := T#100ms, et =>)
      Move(in := #JOB_2_STEP_40, out1 => "Unit1.Em4.ControlNodes".sideTapeAttachment.sequence.status.nextStep)
   END_RUNG
   // the same network as SCL:
   #_w1 := ("Unit1.Em4.ControlNodes".sideTapeAttachment.sequence.status.currentStep = #JOB_2_STEP_31) AND "Unit1.Em4.ControlNodes".sideTapeAttachment.sequence.status.seqActive;
   "Unit1.Em4.ControlNodes".sideTapeAttachment."step".action1[231] := #_w1 AND NOT "Unit1.Em4.ControlNodes".cmSideTapeCutterBwdFwd.monitoring.inHomePos;
   "Unit1.Em4.ControlNodes".sideTapeAttachment."step".transition1[231] := #_w1 AND "Unit1.Em4.ControlNodes".cmSideTapeCutterBwdFwd.monitoring.inHomePos;
   #statTonTime[231].TON(IN := #_w1 AND "Unit1.Em4.ControlNodes".sideTapeAttachment."step".transition1[231],
                         PT := T#100ms);
   IF #statTonTime[231].Q THEN
       "Unit1.Em4.ControlNodes".sideTapeAttachment.sequence.status.nextStep := #JOB_2_STEP_40;
   END_IF;
END_REGION

REGION Network 32: Step[240] : Side Tape Clamp Open
   RUNG wire#powerrail
      { S7_Templates := "SrcType := DInt" } EQ_Contact(in1 := "Unit1.Em4.ControlNodes".sideTapeAttachment.sequence.status.currentStep, in2 := #JOB_2_STEP_40)
      Contact( "Unit1.Em4.ControlNodes".sideTapeAttachment.sequence.status.seqActive )
      wire#w1
      I_Contact( "Unit1.Em4.ControlNodes".cmSideTapeLoadingClampOpenClose.monitoring.inHomePos )
      Coil( "Unit1.Em4.ControlNodes".sideTapeAttachment."step".action1[240] )
   END_RUNG
   RUNG wire#w1
      Contact( "Unit1.Em4.ControlNodes".cmSideTapeLoadingClampOpenClose.monitoring.inHomePos )
      Coil( "Unit1.Em4.ControlNodes".sideTapeAttachment."step".transition1[240] )
   END_RUNG
   RUNG wire#w1
      Contact( "Unit1.Em4.ControlNodes".sideTapeAttachment."step".transition1[240] )
      { S7_Templates := "time_type := Time" } #statTonTime[240].TON(pt := T#100ms, et =>)
      Move(in := #JOB_2_STEP_41, out1 => "Unit1.Em4.ControlNodes".sideTapeAttachment.sequence.status.nextStep)
   END_RUNG
   // the same network as SCL:
   #_w1 := ("Unit1.Em4.ControlNodes".sideTapeAttachment.sequence.status.currentStep = #JOB_2_STEP_40) AND "Unit1.Em4.ControlNodes".sideTapeAttachment.sequence.status.seqActive;
   "Unit1.Em4.ControlNodes".sideTapeAttachment."step".action1[240] := #_w1 AND NOT "Unit1.Em4.ControlNodes".cmSideTapeLoadingClampOpenClose.monitoring.inHomePos;
   "Unit1.Em4.ControlNodes".sideTapeAttachment."step".transition1[240] := #_w1 AND "Unit1.Em4.ControlNodes".cmSideTapeLoadingClampOpenClose.monitoring.inHomePos;
   #statTonTime[240].TON(IN := #_w1 AND "Unit1.Em4.ControlNodes".sideTapeAttachment."step".transition1[240],
                         PT := T#100ms);
   IF #statTonTime[240].Q THEN
       "Unit1.Em4.ControlNodes".sideTapeAttachment.sequence.status.nextStep := #JOB_2_STEP_41;
   END_IF;
END_REGION

REGION Network 33: Step[241] : Spare
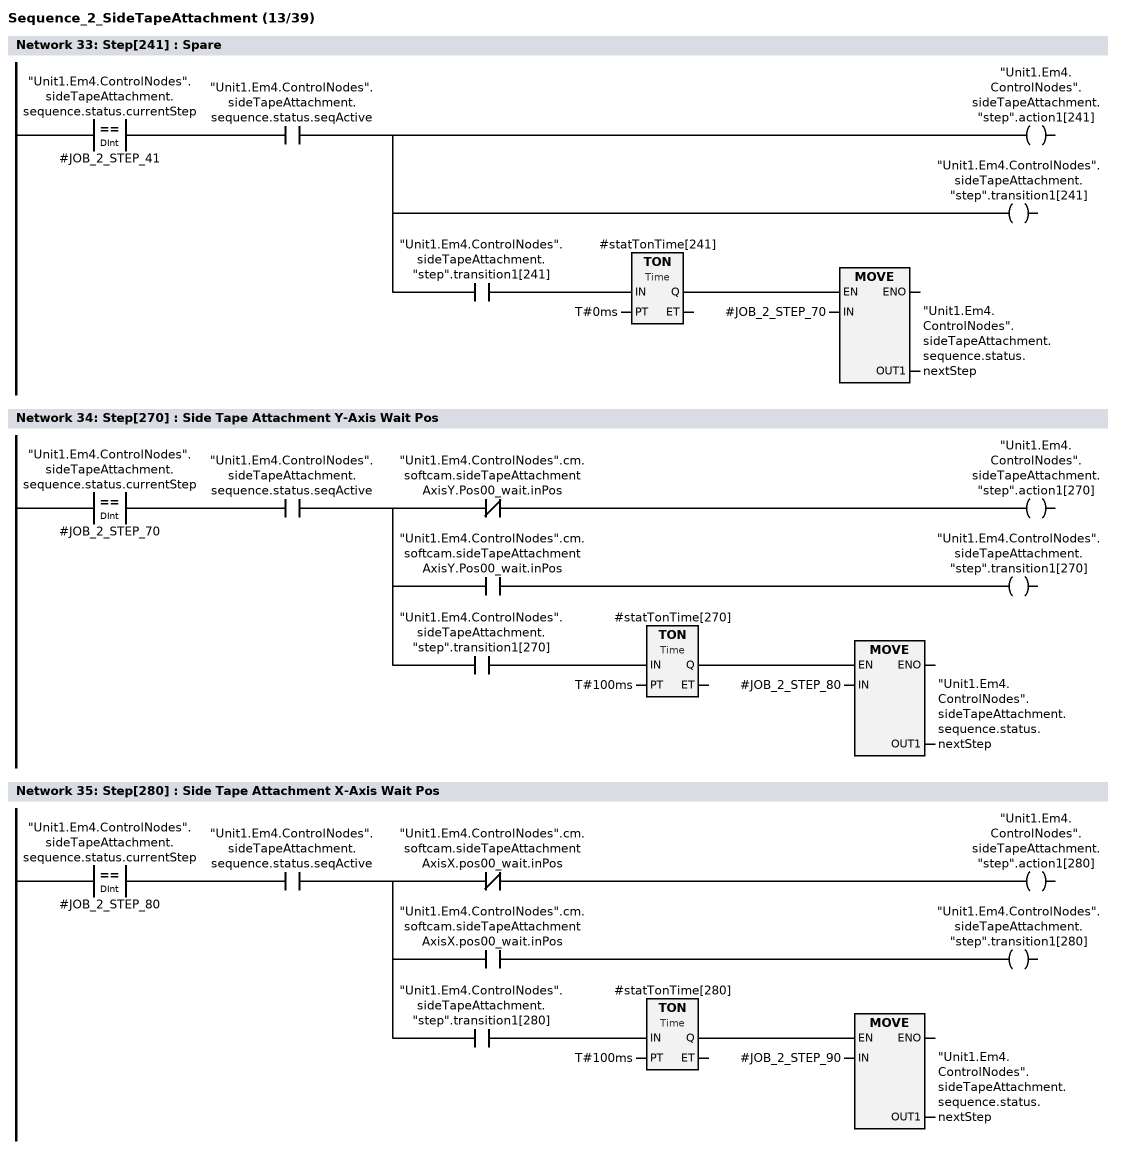
   RUNG wire#powerrail
      { S7_Templates := "SrcType := DInt" } EQ_Contact(in1 := "Unit1.Em4.ControlNodes".sideTapeAttachment.sequence.status.currentStep, in2 := #JOB_2_STEP_41)
      Contact( "Unit1.Em4.ControlNodes".sideTapeAttachment.sequence.status.seqActive )
      wire#w1
      Coil( "Unit1.Em4.ControlNodes".sideTapeAttachment."step".action1[241] )
   END_RUNG
   RUNG wire#w1
      Coil( "Unit1.Em4.ControlNodes".sideTapeAttachment."step".transition1[241] )
   END_RUNG
   RUNG wire#w1
      Contact( "Unit1.Em4.ControlNodes".sideTapeAttachment."step".transition1[241] )
      { S7_Templates := "time_type := Time" } #statTonTime[241].TON(pt := T#0ms, et =>)
      Move(in := #JOB_2_STEP_70, out1 => "Unit1.Em4.ControlNodes".sideTapeAttachment.sequence.status.nextStep)
   END_RUNG
   // the same network as SCL:
   "Unit1.Em4.ControlNodes".sideTapeAttachment."step".action1[241] := ("Unit1.Em4.ControlNodes".sideTapeAttachment.sequence.status.currentStep = #JOB_2_STEP_41) AND "Unit1.Em4.ControlNodes".sideTapeAttachment.sequence.status.seqActive;
   "Unit1.Em4.ControlNodes".sideTapeAttachment."step".transition1[241] := ("Unit1.Em4.ControlNodes".sideTapeAttachment.sequence.status.currentStep = #JOB_2_STEP_41) AND "Unit1.Em4.ControlNodes".sideTapeAttachment.sequence.status.seqActive;
   #statTonTime[241].TON(IN := ("Unit1.Em4.ControlNodes".sideTapeAttachment.sequence.status.currentStep = #JOB_2_STEP_41) AND "Unit1.Em4.ControlNodes".sideTapeAttachment.sequence.status.seqActive AND "Unit1.Em4.ControlNodes".sideTapeAttachment."step".transition1[241],
                         PT := T#0ms);
   IF #statTonTime[241].Q THEN
       "Unit1.Em4.ControlNodes".sideTapeAttachment.sequence.status.nextStep := #JOB_2_STEP_70;
   END_IF;
END_REGION

REGION Network 34: Step[270] : Side Tape Attachment Y-Axis Wait Pos
   RUNG wire#powerrail
      { S7_Templates := "SrcType := DInt" } EQ_Contact(in1 := "Unit1.Em4.ControlNodes".sideTapeAttachment.sequence.status.currentStep, in2 := #JOB_2_STEP_70)
      Contact( "Unit1.Em4.ControlNodes".sideTapeAttachment.sequence.status.seqActive )
      wire#w1
      I_Contact( "Unit1.Em4.ControlNodes".cm.softcam.sideTapeAttachmentAxisY.Pos00_wait.inPos )
      Coil( "Unit1.Em4.ControlNodes".sideTapeAttachment."step".action1[270] )
   END_RUNG
   RUNG wire#w1
      Contact( "Unit1.Em4.ControlNodes".cm.softcam.sideTapeAttachmentAxisY.Pos00_wait.inPos )
      Coil( "Unit1.Em4.ControlNodes".sideTapeAttachment."step".transition1[270] )
   END_RUNG
   RUNG wire#w1
      Contact( "Unit1.Em4.ControlNodes".sideTapeAttachment."step".transition1[270] )
      { S7_Templates := "time_type := Time" } #statTonTime[270].TON(pt := T#100ms, et =>)
      Move(in := #JOB_2_STEP_80, out1 => "Unit1.Em4.ControlNodes".sideTapeAttachment.sequence.status.nextStep)
   END_RUNG
   // the same network as SCL:
   #_w1 := ("Unit1.Em4.ControlNodes".sideTapeAttachment.sequence.status.currentStep = #JOB_2_STEP_70) AND "Unit1.Em4.ControlNodes".sideTapeAttachment.sequence.status.seqActive;
   "Unit1.Em4.ControlNodes".sideTapeAttachment."step".action1[270] := #_w1 AND NOT "Unit1.Em4.ControlNodes".cm.softcam.sideTapeAttachmentAxisY.Pos00_wait.inPos;
   "Unit1.Em4.ControlNodes".sideTapeAttachment."step".transition1[270] := #_w1 AND "Unit1.Em4.ControlNodes".cm.softcam.sideTapeAttachmentAxisY.Pos00_wait.inPos;
   #statTonTime[270].TON(IN := #_w1 AND "Unit1.Em4.ControlNodes".sideTapeAttachment."step".transition1[270],
                         PT := T#100ms);
   IF #statTonTime[270].Q THEN
       "Unit1.Em4.ControlNodes".sideTapeAttachment.sequence.status.nextStep := #JOB_2_STEP_80;
   END_IF;
END_REGION

REGION Network 35: Step[280] : Side Tape Attachment X-Axis Wait Pos
   RUNG wire#powerrail
      { S7_Templates := "SrcType := DInt" } EQ_Contact(in1 := "Unit1.Em4.ControlNodes".sideTapeAttachment.sequence.status.currentStep, in2 := #JOB_2_STEP_80)
      Contact( "Unit1.Em4.ControlNodes".sideTapeAttachment.sequence.status.seqActive )
      wire#w1
      I_Contact( "Unit1.Em4.ControlNodes".cm.softcam.sideTapeAttachmentAxisX.pos00_wait.inPos )
      Coil( "Unit1.Em4.ControlNodes".sideTapeAttachment."step".action1[280] )
   END_RUNG
   RUNG wire#w1
      Contact( "Unit1.Em4.ControlNodes".cm.softcam.sideTapeAttachmentAxisX.pos00_wait.inPos )
      Coil( "Unit1.Em4.ControlNodes".sideTapeAttachment."step".transition1[280] )
   END_RUNG
   RUNG wire#w1
      Contact( "Unit1.Em4.ControlNodes".sideTapeAttachment."step".transition1[280] )
      { S7_Templates := "time_type := Time" } #statTonTime[280].TON(pt := T#100ms, et =>)
      Move(in := #JOB_2_STEP_90, out1 => "Unit1.Em4.ControlNodes".sideTapeAttachment.sequence.status.nextStep)
   END_RUNG
   // the same network as SCL:
   #_w1 := ("Unit1.Em4.ControlNodes".sideTapeAttachment.sequence.status.currentStep = #JOB_2_STEP_80) AND "Unit1.Em4.ControlNodes".sideTapeAttachment.sequence.status.seqActive;
   "Unit1.Em4.ControlNodes".sideTapeAttachment."step".action1[280] := #_w1 AND NOT "Unit1.Em4.ControlNodes".cm.softcam.sideTapeAttachmentAxisX.pos00_wait.inPos;
   "Unit1.Em4.ControlNodes".sideTapeAttachment."step".transition1[280] := #_w1 AND "Unit1.Em4.ControlNodes".cm.softcam.sideTapeAttachmentAxisX.pos00_wait.inPos;
   #statTonTime[280].TON(IN := #_w1 AND "Unit1.Em4.ControlNodes".sideTapeAttachment."step".transition1[280],
                         PT := T#100ms);
   IF #statTonTime[280].Q THEN
       "Unit1.Em4.ControlNodes".sideTapeAttachment.sequence.status.nextStep := #JOB_2_STEP_90;
   END_IF;
END_REGION

REGION Network 36: Step[290] : Job[2] Step End
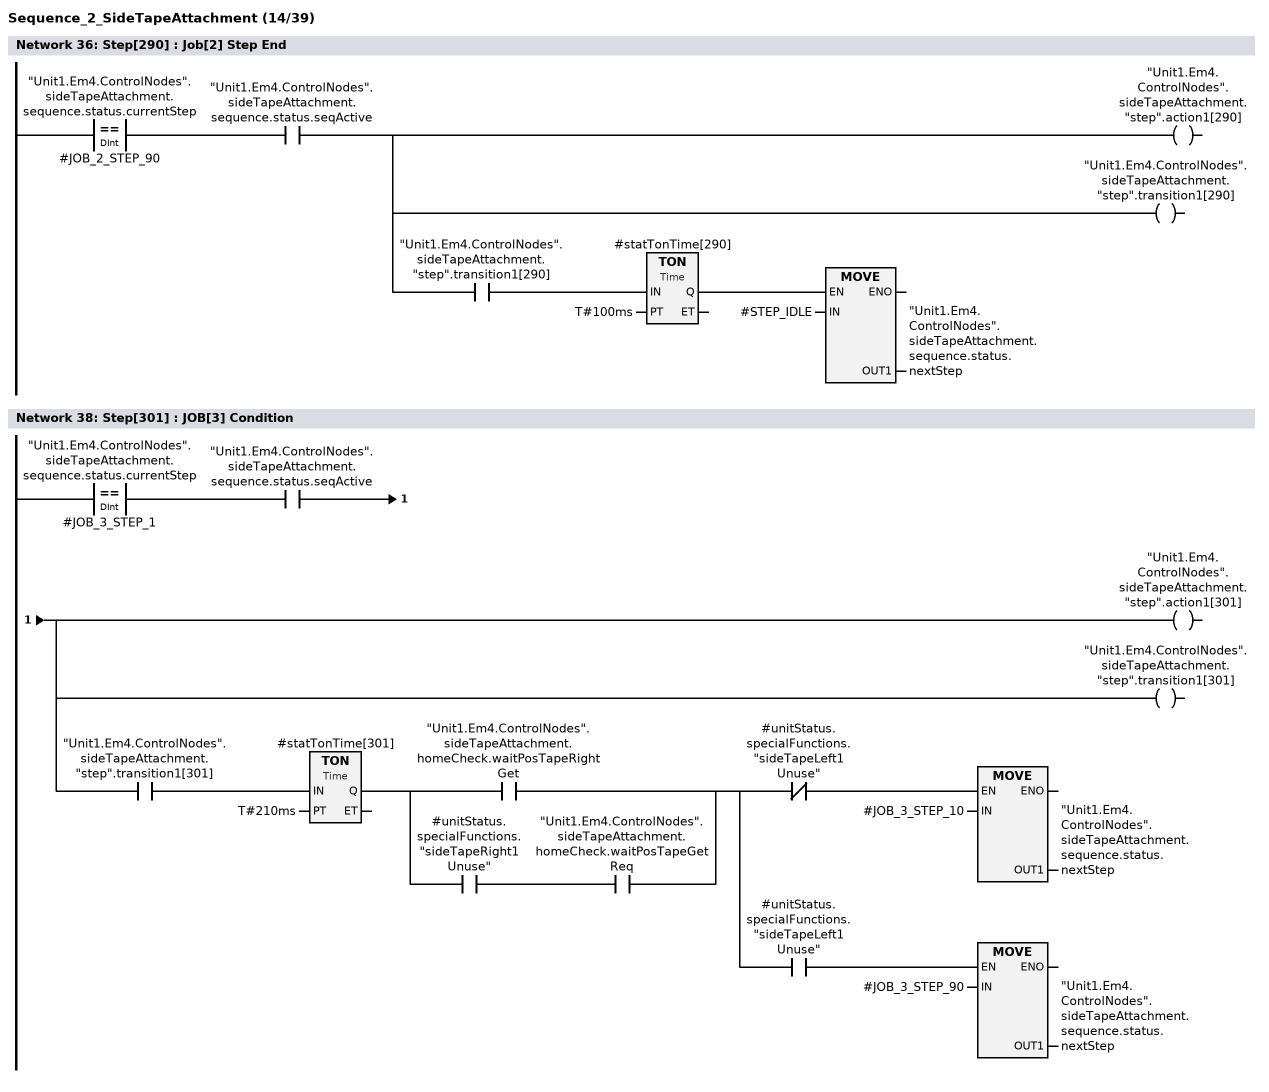
   RUNG wire#powerrail
      { S7_Templates := "SrcType := DInt" } EQ_Contact(in1 := "Unit1.Em4.ControlNodes".sideTapeAttachment.sequence.status.currentStep, in2 := #JOB_2_STEP_90)
      Contact( "Unit1.Em4.ControlNodes".sideTapeAttachment.sequence.status.seqActive )
      wire#w1
      Coil( "Unit1.Em4.ControlNodes".sideTapeAttachment."step".action1[290] )
   END_RUNG
   RUNG wire#w1
      Coil( "Unit1.Em4.ControlNodes".sideTapeAttachment."step".transition1[290] )
   END_RUNG
   RUNG wire#w1
      Contact( "Unit1.Em4.ControlNodes".sideTapeAttachment."step".transition1[290] )
      { S7_Templates := "time_type := Time" } #statTonTime[290].TON(pt := T#100ms, et =>)
      Move(in := #STEP_IDLE, out1 => "Unit1.Em4.ControlNodes".sideTapeAttachment.sequence.status.nextStep)
   END_RUNG
   // the same network as SCL:
   "Unit1.Em4.ControlNodes".sideTapeAttachment."step".action1[290] := ("Unit1.Em4.ControlNodes".sideTapeAttachment.sequence.status.currentStep = #JOB_2_STEP_90) AND "Unit1.Em4.ControlNodes".sideTapeAttachment.sequence.status.seqActive;
   "Unit1.Em4.ControlNodes".sideTapeAttachment."step".transition1[290] := ("Unit1.Em4.ControlNodes".sideTapeAttachment.sequence.status.currentStep = #JOB_2_STEP_90) AND "Unit1.Em4.ControlNodes".sideTapeAttachment.sequence.status.seqActive;
   #statTonTime[290].TON(IN := ("Unit1.Em4.ControlNodes".sideTapeAttachment.sequence.status.currentStep = #JOB_2_STEP_90) AND "Unit1.Em4.ControlNodes".sideTapeAttachment.sequence.status.seqActive AND "Unit1.Em4.ControlNodes".sideTapeAttachment."step".transition1[290],
                         PT := T#100ms);
   IF #statTonTime[290].Q THEN
       "Unit1.Em4.ControlNodes".sideTapeAttachment.sequence.status.nextStep := #STEP_IDLE;
   END_IF;
END_REGION

REGION Network 37: *************** JOB[3] SIDE TAPE LEFT GET=AUTO *************************
END_REGION

REGION Network 38: Step[301] : JOB[3] Condition
   RUNG wire#powerrail
      { S7_Templates := "SrcType := DInt" } EQ_Contact(in1 := "Unit1.Em4.ControlNodes".sideTapeAttachment.sequence.status.currentStep, in2 := #JOB_3_STEP_1)
      Contact( "Unit1.Em4.ControlNodes".sideTapeAttachment.sequence.status.seqActive )
      wire#w1
      Coil( "Unit1.Em4.ControlNodes".sideTapeAttachment."step".action1[301] )
   END_RUNG
   RUNG wire#w1
      Coil( "Unit1.Em4.ControlNodes".sideTapeAttachment."step".transition1[301] )
   END_RUNG
   RUNG wire#w1
      Contact( "Unit1.Em4.ControlNodes".sideTapeAttachment."step".transition1[301] )
      { S7_Templates := "time_type := Time" } #statTonTime[301].TON(pt := T#210ms, et =>)
      wire#w2
      Contact( "Unit1.Em4.ControlNodes".sideTapeAttachment.homeCheck.waitPosTapeRightGet )
      wire#w3
      I_Contact( #unitStatus.specialFunctions."sideTapeLeft1 Unuse" )
      Move(in := #JOB_3_STEP_10, out1 => "Unit1.Em4.ControlNodes".sideTapeAttachment.sequence.status.nextStep)
   END_RUNG
   RUNG wire#w2
      Contact( #unitStatus.specialFunctions."sideTapeRight1 Unuse" )
      Contact( "Unit1.Em4.ControlNodes".sideTapeAttachment.homeCheck.waitPosTapeGetReq )
   END_RUNG wire#w3
   RUNG wire#w3
      Contact( #unitStatus.specialFunctions."sideTapeLeft1 Unuse" )
      Move(in := #JOB_3_STEP_90, out1 => "Unit1.Em4.ControlNodes".sideTapeAttachment.sequence.status.nextStep)
   END_RUNG
   // the same network as SCL:
   "Unit1.Em4.ControlNodes".sideTapeAttachment."step".action1[301] := ("Unit1.Em4.ControlNodes".sideTapeAttachment.sequence.status.currentStep = #JOB_3_STEP_1) AND "Unit1.Em4.ControlNodes".sideTapeAttachment.sequence.status.seqActive;
   "Unit1.Em4.ControlNodes".sideTapeAttachment."step".transition1[301] := ("Unit1.Em4.ControlNodes".sideTapeAttachment.sequence.status.currentStep = #JOB_3_STEP_1) AND "Unit1.Em4.ControlNodes".sideTapeAttachment.sequence.status.seqActive;
   #statTonTime[301].TON(IN := ("Unit1.Em4.ControlNodes".sideTapeAttachment.sequence.status.currentStep = #JOB_3_STEP_1) AND "Unit1.Em4.ControlNodes".sideTapeAttachment.sequence.status.seqActive AND "Unit1.Em4.ControlNodes".sideTapeAttachment."step".transition1[301],
                         PT := T#210ms);
   #_w1 := #statTonTime[301].Q AND ("Unit1.Em4.ControlNodes".sideTapeAttachment.homeCheck.waitPosTapeRightGet OR (#unitStatus.specialFunctions."sideTapeRight1 Unuse" AND "Unit1.Em4.ControlNodes".sideTapeAttachment.homeCheck.waitPosTapeGetReq));
   IF #_w1 AND NOT #unitStatus.specialFunctions."sideTapeLeft1 Unuse" THEN
       "Unit1.Em4.ControlNodes".sideTapeAttachment.sequence.status.nextStep := #JOB_3_STEP_10;
   END_IF;
   IF #_w1 AND #unitStatus.specialFunctions."sideTapeLeft1 Unuse" THEN
       "Unit1.Em4.ControlNodes".sideTapeAttachment.sequence.status.nextStep := #JOB_3_STEP_90;
   END_IF;
END_REGION

REGION Network 39: Step[310] : Side Tape Attachment X-Axis Left Tape Get Pos
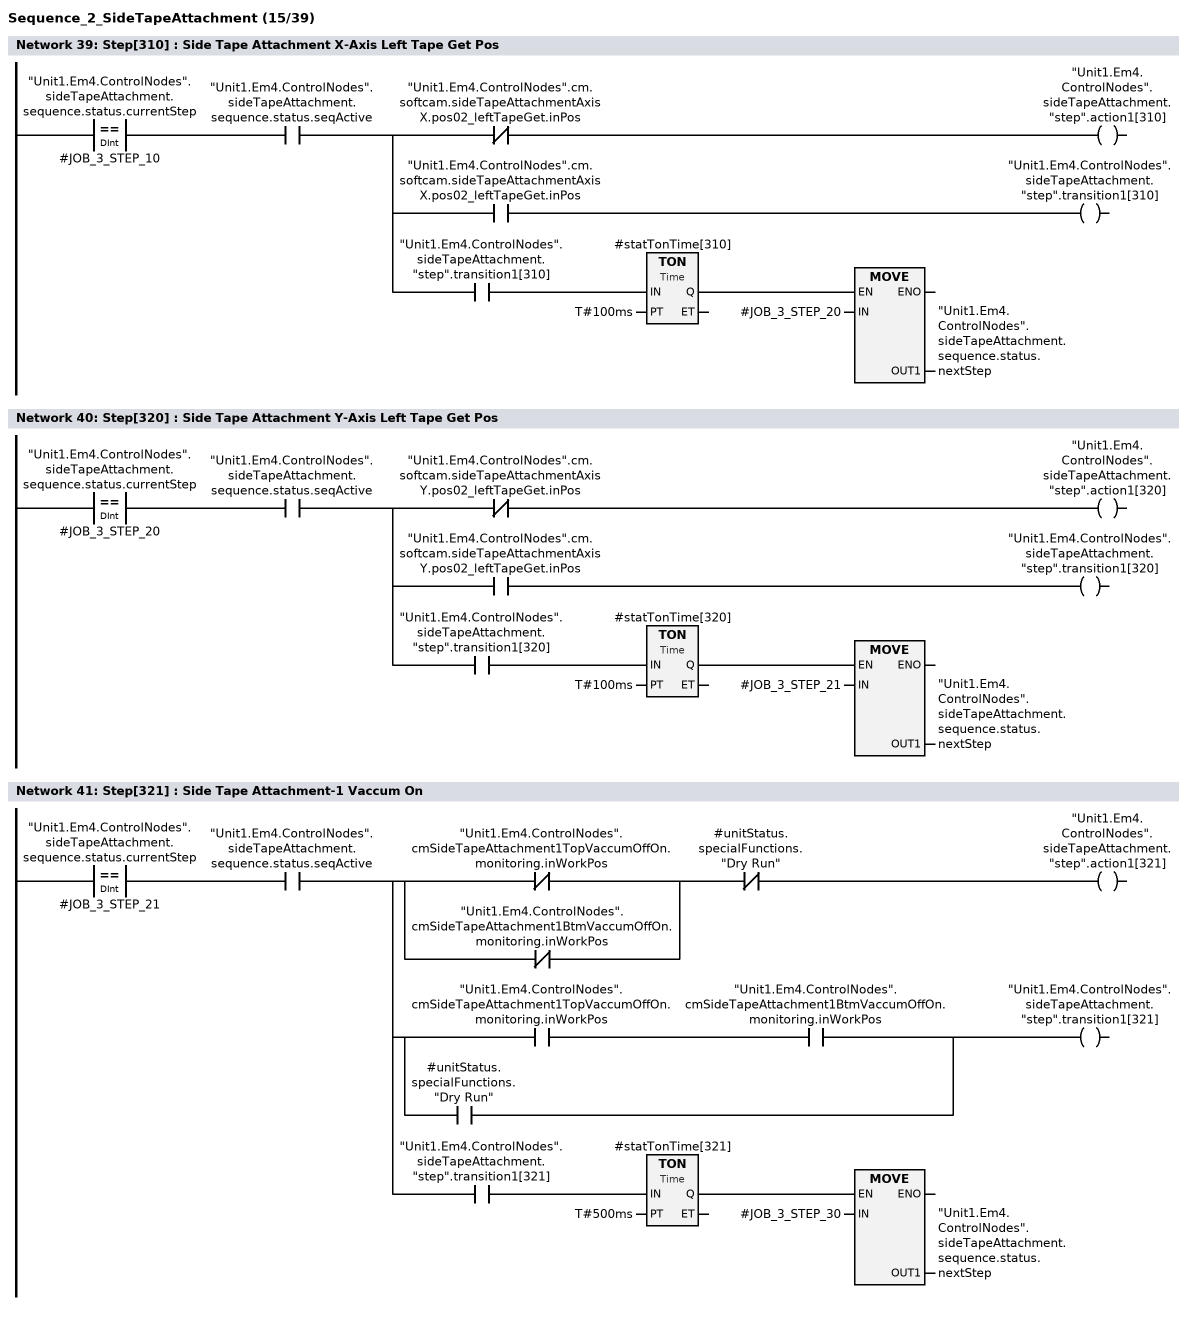
   RUNG wire#powerrail
      { S7_Templates := "SrcType := DInt" } EQ_Contact(in1 := "Unit1.Em4.ControlNodes".sideTapeAttachment.sequence.status.currentStep, in2 := #JOB_3_STEP_10)
      Contact( "Unit1.Em4.ControlNodes".sideTapeAttachment.sequence.status.seqActive )
      wire#w1
      I_Contact( "Unit1.Em4.ControlNodes".cm.softcam.sideTapeAttachmentAxisX.pos02_leftTapeGet.inPos )
      Coil( "Unit1.Em4.ControlNodes".sideTapeAttachment."step".action1[310] )
   END_RUNG
   RUNG wire#w1
      Contact( "Unit1.Em4.ControlNodes".cm.softcam.sideTapeAttachmentAxisX.pos02_leftTapeGet.inPos )
      Coil( "Unit1.Em4.ControlNodes".sideTapeAttachment."step".transition1[310] )
   END_RUNG
   RUNG wire#w1
      Contact( "Unit1.Em4.ControlNodes".sideTapeAttachment."step".transition1[310] )
      { S7_Templates := "time_type := Time" } #statTonTime[310].TON(pt := T#100ms, et =>)
      Move(in := #JOB_3_STEP_20, out1 => "Unit1.Em4.ControlNodes".sideTapeAttachment.sequence.status.nextStep)
   END_RUNG
   // the same network as SCL:
   #_w1 := ("Unit1.Em4.ControlNodes".sideTapeAttachment.sequence.status.currentStep = #JOB_3_STEP_10) AND "Unit1.Em4.ControlNodes".sideTapeAttachment.sequence.status.seqActive;
   "Unit1.Em4.ControlNodes".sideTapeAttachment."step".action1[310] := #_w1 AND NOT "Unit1.Em4.ControlNodes".cm.softcam.sideTapeAttachmentAxisX.pos02_leftTapeGet.inPos;
   "Unit1.Em4.ControlNodes".sideTapeAttachment."step".transition1[310] := #_w1 AND "Unit1.Em4.ControlNodes".cm.softcam.sideTapeAttachmentAxisX.pos02_leftTapeGet.inPos;
   #statTonTime[310].TON(IN := #_w1 AND "Unit1.Em4.ControlNodes".sideTapeAttachment."step".transition1[310],
                         PT := T#100ms);
   IF #statTonTime[310].Q THEN
       "Unit1.Em4.ControlNodes".sideTapeAttachment.sequence.status.nextStep := #JOB_3_STEP_20;
   END_IF;
END_REGION

REGION Network 40: Step[320] : Side Tape Attachment Y-Axis Left Tape Get Pos
   RUNG wire#powerrail
      { S7_Templates := "SrcType := DInt" } EQ_Contact(in1 := "Unit1.Em4.ControlNodes".sideTapeAttachment.sequence.status.currentStep, in2 := #JOB_3_STEP_20)
      Contact( "Unit1.Em4.ControlNodes".sideTapeAttachment.sequence.status.seqActive )
      wire#w1
      I_Contact( "Unit1.Em4.ControlNodes".cm.softcam.sideTapeAttachmentAxisY.pos02_leftTapeGet.inPos )
      Coil( "Unit1.Em4.ControlNodes".sideTapeAttachment."step".action1[320] )
   END_RUNG
   RUNG wire#w1
      Contact( "Unit1.Em4.ControlNodes".cm.softcam.sideTapeAttachmentAxisY.pos02_leftTapeGet.inPos )
      Coil( "Unit1.Em4.ControlNodes".sideTapeAttachment."step".transition1[320] )
   END_RUNG
   RUNG wire#w1
      Contact( "Unit1.Em4.ControlNodes".sideTapeAttachment."step".transition1[320] )
      { S7_Templates := "time_type := Time" } #statTonTime[320].TON(pt := T#100ms, et =>)
      Move(in := #JOB_3_STEP_21, out1 => "Unit1.Em4.ControlNodes".sideTapeAttachment.sequence.status.nextStep)
   END_RUNG
   // the same network as SCL:
   #_w1 := ("Unit1.Em4.ControlNodes".sideTapeAttachment.sequence.status.currentStep = #JOB_3_STEP_20) AND "Unit1.Em4.ControlNodes".sideTapeAttachment.sequence.status.seqActive;
   "Unit1.Em4.ControlNodes".sideTapeAttachment."step".action1[320] := #_w1 AND NOT "Unit1.Em4.ControlNodes".cm.softcam.sideTapeAttachmentAxisY.pos02_leftTapeGet.inPos;
   "Unit1.Em4.ControlNodes".sideTapeAttachment."step".transition1[320] := #_w1 AND "Unit1.Em4.ControlNodes".cm.softcam.sideTapeAttachmentAxisY.pos02_leftTapeGet.inPos;
   #statTonTime[320].TON(IN := #_w1 AND "Unit1.Em4.ControlNodes".sideTapeAttachment."step".transition1[320],
                         PT := T#100ms);
   IF #statTonTime[320].Q THEN
       "Unit1.Em4.ControlNodes".sideTapeAttachment.sequence.status.nextStep := #JOB_3_STEP_21;
   END_IF;
END_REGION

REGION Network 41: Step[321] : Side Tape Attachment-1 Vaccum On
   RUNG wire#powerrail
      { S7_Templates := "SrcType := DInt" } EQ_Contact(in1 := "Unit1.Em4.ControlNodes".sideTapeAttachment.sequence.status.currentStep, in2 := #JOB_3_STEP_21)
      Contact( "Unit1.Em4.ControlNodes".sideTapeAttachment.sequence.status.seqActive )
      wire#w1
      I_Contact( "Unit1.Em4.ControlNodes".cmSideTapeAttachment1TopVaccumOffOn.monitoring.inWorkPos )
      wire#w2
      I_Contact( #unitStatus.specialFunctions."Dry Run" )
      Coil( "Unit1.Em4.ControlNodes".sideTapeAttachment."step".action1[321] )
   END_RUNG
   RUNG wire#w1
      I_Contact( "Unit1.Em4.ControlNodes".cmSideTapeAttachment1BtmVaccumOffOn.monitoring.inWorkPos )
   END_RUNG wire#w2
   RUNG wire#w1
      Contact( "Unit1.Em4.ControlNodes".cmSideTapeAttachment1TopVaccumOffOn.monitoring.inWorkPos )
      Contact( "Unit1.Em4.ControlNodes".cmSideTapeAttachment1BtmVaccumOffOn.monitoring.inWorkPos )
      wire#w3
      Coil( "Unit1.Em4.ControlNodes".sideTapeAttachment."step".transition1[321] )
   END_RUNG
   RUNG wire#w1
      Contact( #unitStatus.specialFunctions."Dry Run" )
   END_RUNG wire#w3
   RUNG wire#w1
      Contact( "Unit1.Em4.ControlNodes".sideTapeAttachment."step".transition1[321] )
      { S7_Templates := "time_type := Time" } #statTonTime[321].TON(pt := T#500ms, et =>)
      Move(in := #JOB_3_STEP_30, out1 => "Unit1.Em4.ControlNodes".sideTapeAttachment.sequence.status.nextStep)
   END_RUNG
   // the same network as SCL:
   #_w1 := ("Unit1.Em4.ControlNodes".sideTapeAttachment.sequence.status.currentStep = #JOB_3_STEP_21) AND "Unit1.Em4.ControlNodes".sideTapeAttachment.sequence.status.seqActive;
   "Unit1.Em4.ControlNodes".sideTapeAttachment."step".action1[321] := #_w1 AND (NOT "Unit1.Em4.ControlNodes".cmSideTapeAttachment1TopVaccumOffOn.monitoring.inWorkPos OR NOT "Unit1.Em4.ControlNodes".cmSideTapeAttachment1BtmVaccumOffOn.monitoring.inWorkPos) AND NOT #unitStatus.specialFunctions."Dry Run";
   "Unit1.Em4.ControlNodes".sideTapeAttachment."step".transition1[321] := #_w1 AND (("Unit1.Em4.ControlNodes".cmSideTapeAttachment1TopVaccumOffOn.monitoring.inWorkPos AND "Unit1.Em4.ControlNodes".cmSideTapeAttachment1BtmVaccumOffOn.monitoring.inWorkPos) OR #unitStatus.specialFunctions."Dry Run");
   #statTonTime[321].TON(IN := #_w1 AND "Unit1.Em4.ControlNodes".sideTapeAttachment."step".transition1[321],
                         PT := T#500ms);
   IF #statTonTime[321].Q THEN
       "Unit1.Em4.ControlNodes".sideTapeAttachment.sequence.status.nextStep := #JOB_3_STEP_30;
   END_IF;
END_REGION

REGION Network 42: Step[330] : Side Tape Cutter Forward
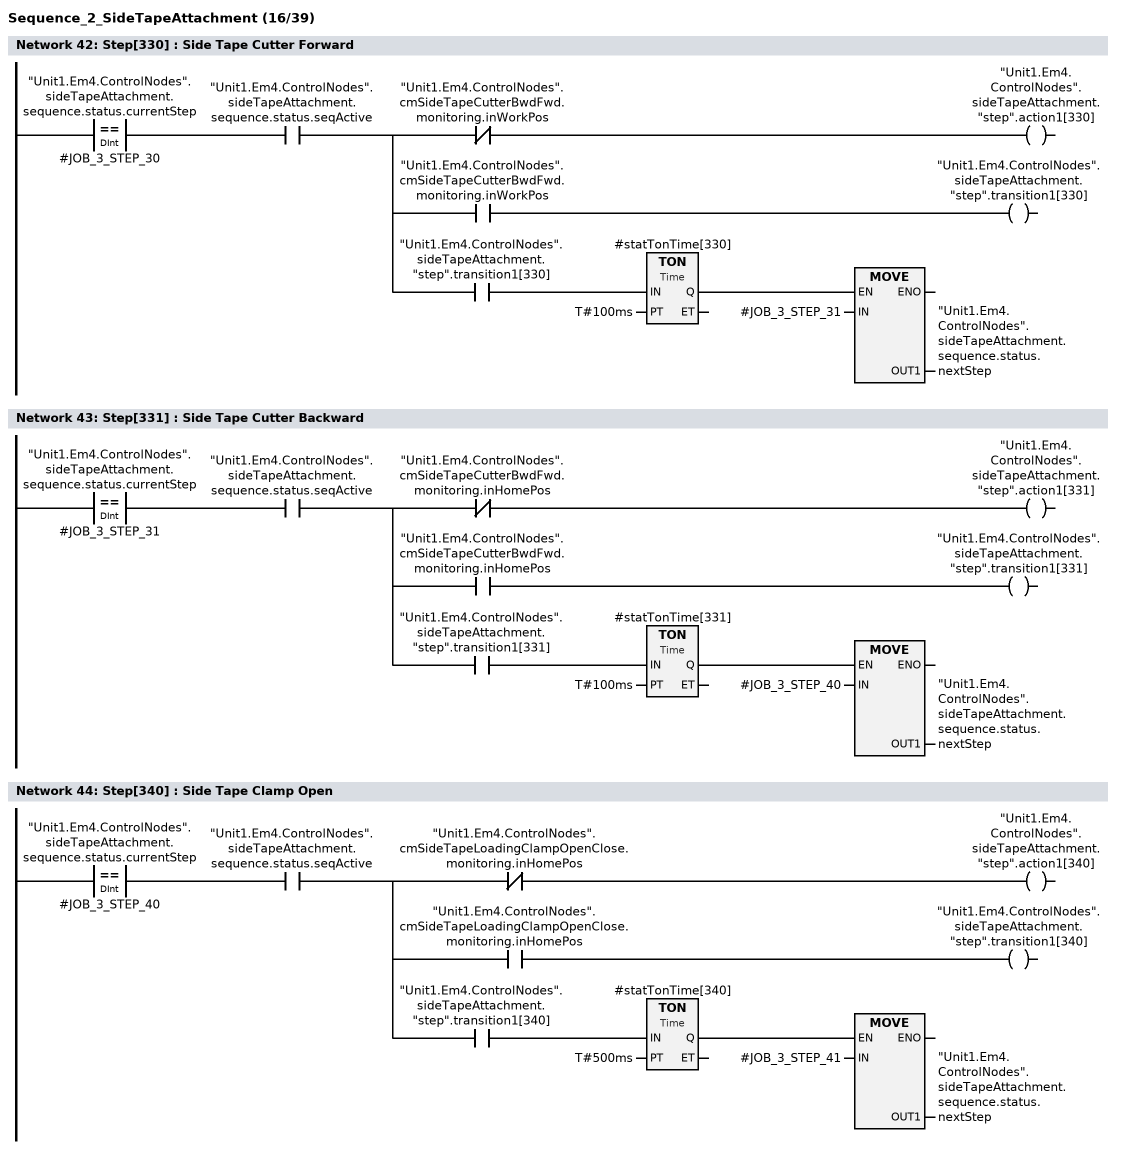
   RUNG wire#powerrail
      { S7_Templates := "SrcType := DInt" } EQ_Contact(in1 := "Unit1.Em4.ControlNodes".sideTapeAttachment.sequence.status.currentStep, in2 := #JOB_3_STEP_30)
      Contact( "Unit1.Em4.ControlNodes".sideTapeAttachment.sequence.status.seqActive )
      wire#w1
      I_Contact( "Unit1.Em4.ControlNodes".cmSideTapeCutterBwdFwd.monitoring.inWorkPos )
      Coil( "Unit1.Em4.ControlNodes".sideTapeAttachment."step".action1[330] )
   END_RUNG
   RUNG wire#w1
      Contact( "Unit1.Em4.ControlNodes".cmSideTapeCutterBwdFwd.monitoring.inWorkPos )
      Coil( "Unit1.Em4.ControlNodes".sideTapeAttachment."step".transition1[330] )
   END_RUNG
   RUNG wire#w1
      Contact( "Unit1.Em4.ControlNodes".sideTapeAttachment."step".transition1[330] )
      { S7_Templates := "time_type := Time" } #statTonTime[330].TON(pt := T#100ms, et =>)
      Move(in := #JOB_3_STEP_31, out1 => "Unit1.Em4.ControlNodes".sideTapeAttachment.sequence.status.nextStep)
   END_RUNG
   // the same network as SCL:
   #_w1 := ("Unit1.Em4.ControlNodes".sideTapeAttachment.sequence.status.currentStep = #JOB_3_STEP_30) AND "Unit1.Em4.ControlNodes".sideTapeAttachment.sequence.status.seqActive;
   "Unit1.Em4.ControlNodes".sideTapeAttachment."step".action1[330] := #_w1 AND NOT "Unit1.Em4.ControlNodes".cmSideTapeCutterBwdFwd.monitoring.inWorkPos;
   "Unit1.Em4.ControlNodes".sideTapeAttachment."step".transition1[330] := #_w1 AND "Unit1.Em4.ControlNodes".cmSideTapeCutterBwdFwd.monitoring.inWorkPos;
   #statTonTime[330].TON(IN := #_w1 AND "Unit1.Em4.ControlNodes".sideTapeAttachment."step".transition1[330],
                         PT := T#100ms);
   IF #statTonTime[330].Q THEN
       "Unit1.Em4.ControlNodes".sideTapeAttachment.sequence.status.nextStep := #JOB_3_STEP_31;
   END_IF;
END_REGION

REGION Network 43: Step[331] : Side Tape Cutter Backward
   RUNG wire#powerrail
      { S7_Templates := "SrcType := DInt" } EQ_Contact(in1 := "Unit1.Em4.ControlNodes".sideTapeAttachment.sequence.status.currentStep, in2 := #JOB_3_STEP_31)
      Contact( "Unit1.Em4.ControlNodes".sideTapeAttachment.sequence.status.seqActive )
      wire#w1
      I_Contact( "Unit1.Em4.ControlNodes".cmSideTapeCutterBwdFwd.monitoring.inHomePos )
      Coil( "Unit1.Em4.ControlNodes".sideTapeAttachment."step".action1[331] )
   END_RUNG
   RUNG wire#w1
      Contact( "Unit1.Em4.ControlNodes".cmSideTapeCutterBwdFwd.monitoring.inHomePos )
      Coil( "Unit1.Em4.ControlNodes".sideTapeAttachment."step".transition1[331] )
   END_RUNG
   RUNG wire#w1
      Contact( "Unit1.Em4.ControlNodes".sideTapeAttachment."step".transition1[331] )
      { S7_Templates := "time_type := Time" } #statTonTime[331].TON(pt := T#100ms, et =>)
      Move(in := #JOB_3_STEP_40, out1 => "Unit1.Em4.ControlNodes".sideTapeAttachment.sequence.status.nextStep)
   END_RUNG
   // the same network as SCL:
   #_w1 := ("Unit1.Em4.ControlNodes".sideTapeAttachment.sequence.status.currentStep = #JOB_3_STEP_31) AND "Unit1.Em4.ControlNodes".sideTapeAttachment.sequence.status.seqActive;
   "Unit1.Em4.ControlNodes".sideTapeAttachment."step".action1[331] := #_w1 AND NOT "Unit1.Em4.ControlNodes".cmSideTapeCutterBwdFwd.monitoring.inHomePos;
   "Unit1.Em4.ControlNodes".sideTapeAttachment."step".transition1[331] := #_w1 AND "Unit1.Em4.ControlNodes".cmSideTapeCutterBwdFwd.monitoring.inHomePos;
   #statTonTime[331].TON(IN := #_w1 AND "Unit1.Em4.ControlNodes".sideTapeAttachment."step".transition1[331],
                         PT := T#100ms);
   IF #statTonTime[331].Q THEN
       "Unit1.Em4.ControlNodes".sideTapeAttachment.sequence.status.nextStep := #JOB_3_STEP_40;
   END_IF;
END_REGION

REGION Network 44: Step[340] : Side Tape Clamp Open
   RUNG wire#powerrail
      { S7_Templates := "SrcType := DInt" } EQ_Contact(in1 := "Unit1.Em4.ControlNodes".sideTapeAttachment.sequence.status.currentStep, in2 := #JOB_3_STEP_40)
      Contact( "Unit1.Em4.ControlNodes".sideTapeAttachment.sequence.status.seqActive )
      wire#w1
      I_Contact( "Unit1.Em4.ControlNodes".cmSideTapeLoadingClampOpenClose.monitoring.inHomePos )
      Coil( "Unit1.Em4.ControlNodes".sideTapeAttachment."step".action1[340] )
   END_RUNG
   RUNG wire#w1
      Contact( "Unit1.Em4.ControlNodes".cmSideTapeLoadingClampOpenClose.monitoring.inHomePos )
      Coil( "Unit1.Em4.ControlNodes".sideTapeAttachment."step".transition1[340] )
   END_RUNG
   RUNG wire#w1
      Contact( "Unit1.Em4.ControlNodes".sideTapeAttachment."step".transition1[340] )
      { S7_Templates := "time_type := Time" } #statTonTime[340].TON(pt := T#500ms, et =>)
      Move(in := #JOB_3_STEP_41, out1 => "Unit1.Em4.ControlNodes".sideTapeAttachment.sequence.status.nextStep)
   END_RUNG
   // the same network as SCL:
   #_w1 := ("Unit1.Em4.ControlNodes".sideTapeAttachment.sequence.status.currentStep = #JOB_3_STEP_40) AND "Unit1.Em4.ControlNodes".sideTapeAttachment.sequence.status.seqActive;
   "Unit1.Em4.ControlNodes".sideTapeAttachment."step".action1[340] := #_w1 AND NOT "Unit1.Em4.ControlNodes".cmSideTapeLoadingClampOpenClose.monitoring.inHomePos;
   "Unit1.Em4.ControlNodes".sideTapeAttachment."step".transition1[340] := #_w1 AND "Unit1.Em4.ControlNodes".cmSideTapeLoadingClampOpenClose.monitoring.inHomePos;
   #statTonTime[340].TON(IN := #_w1 AND "Unit1.Em4.ControlNodes".sideTapeAttachment."step".transition1[340],
                         PT := T#500ms);
   IF #statTonTime[340].Q THEN
       "Unit1.Em4.ControlNodes".sideTapeAttachment.sequence.status.nextStep := #JOB_3_STEP_41;
   END_IF;
END_REGION

REGION Network 45: Step[341] : Spare
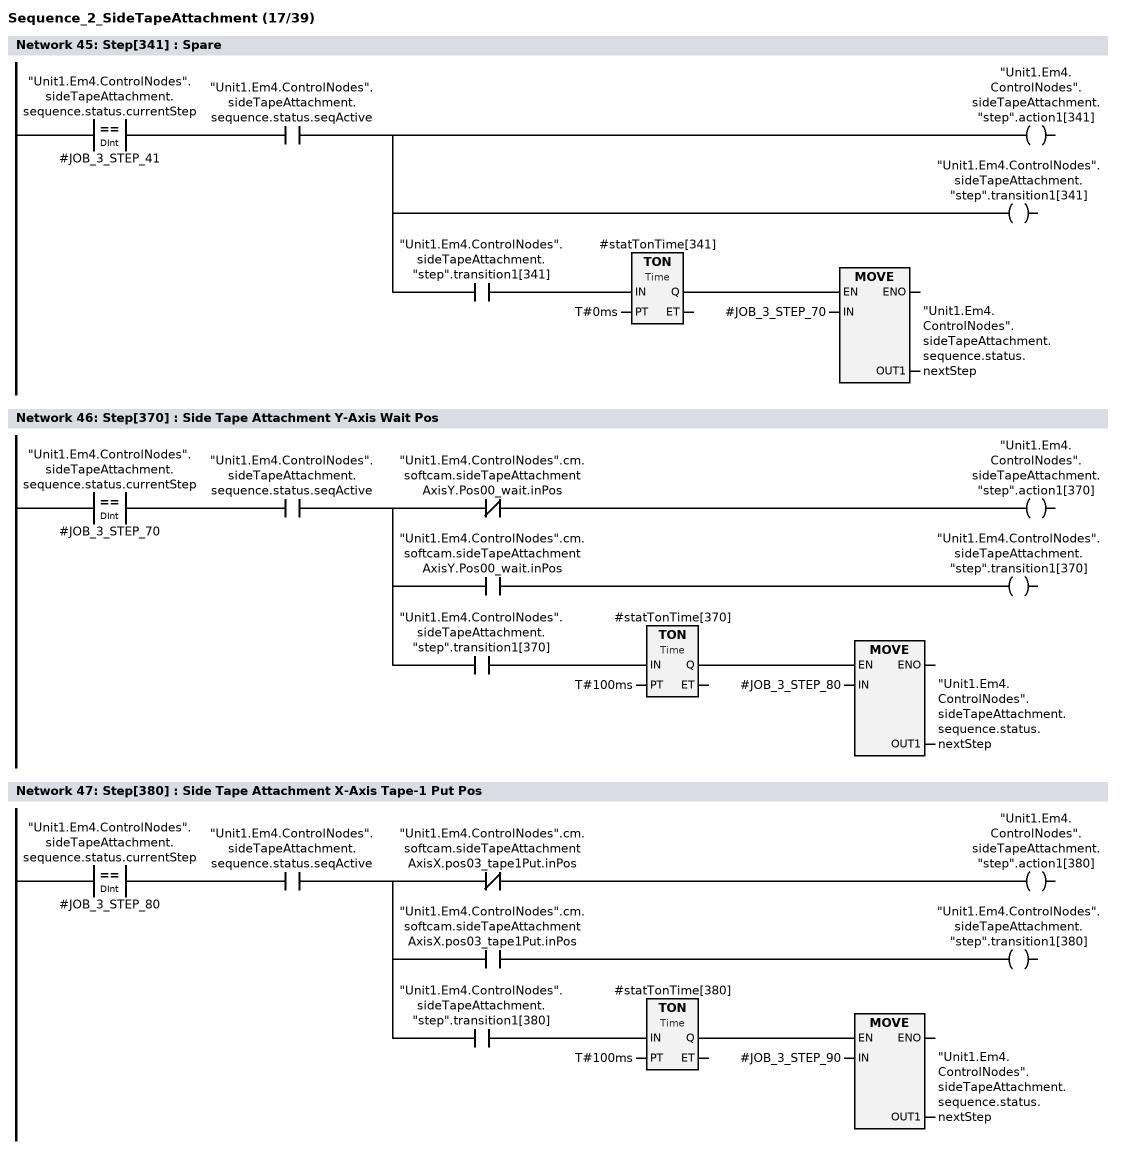
   RUNG wire#powerrail
      { S7_Templates := "SrcType := DInt" } EQ_Contact(in1 := "Unit1.Em4.ControlNodes".sideTapeAttachment.sequence.status.currentStep, in2 := #JOB_3_STEP_41)
      Contact( "Unit1.Em4.ControlNodes".sideTapeAttachment.sequence.status.seqActive )
      wire#w1
      Coil( "Unit1.Em4.ControlNodes".sideTapeAttachment."step".action1[341] )
   END_RUNG
   RUNG wire#w1
      Coil( "Unit1.Em4.ControlNodes".sideTapeAttachment."step".transition1[341] )
   END_RUNG
   RUNG wire#w1
      Contact( "Unit1.Em4.ControlNodes".sideTapeAttachment."step".transition1[341] )
      { S7_Templates := "time_type := Time" } #statTonTime[341].TON(pt := T#0ms, et =>)
      Move(in := #JOB_3_STEP_70, out1 => "Unit1.Em4.ControlNodes".sideTapeAttachment.sequence.status.nextStep)
   END_RUNG
   // the same network as SCL:
   "Unit1.Em4.ControlNodes".sideTapeAttachment."step".action1[341] := ("Unit1.Em4.ControlNodes".sideTapeAttachment.sequence.status.currentStep = #JOB_3_STEP_41) AND "Unit1.Em4.ControlNodes".sideTapeAttachment.sequence.status.seqActive;
   "Unit1.Em4.ControlNodes".sideTapeAttachment."step".transition1[341] := ("Unit1.Em4.ControlNodes".sideTapeAttachment.sequence.status.currentStep = #JOB_3_STEP_41) AND "Unit1.Em4.ControlNodes".sideTapeAttachment.sequence.status.seqActive;
   #statTonTime[341].TON(IN := ("Unit1.Em4.ControlNodes".sideTapeAttachment.sequence.status.currentStep = #JOB_3_STEP_41) AND "Unit1.Em4.ControlNodes".sideTapeAttachment.sequence.status.seqActive AND "Unit1.Em4.ControlNodes".sideTapeAttachment."step".transition1[341],
                         PT := T#0ms);
   IF #statTonTime[341].Q THEN
       "Unit1.Em4.ControlNodes".sideTapeAttachment.sequence.status.nextStep := #JOB_3_STEP_70;
   END_IF;
END_REGION

REGION Network 46: Step[370] : Side Tape Attachment Y-Axis Wait Pos
   RUNG wire#powerrail
      { S7_Templates := "SrcType := DInt" } EQ_Contact(in1 := "Unit1.Em4.ControlNodes".sideTapeAttachment.sequence.status.currentStep, in2 := #JOB_3_STEP_70)
      Contact( "Unit1.Em4.ControlNodes".sideTapeAttachment.sequence.status.seqActive )
      wire#w1
      I_Contact( "Unit1.Em4.ControlNodes".cm.softcam.sideTapeAttachmentAxisY.Pos00_wait.inPos )
      Coil( "Unit1.Em4.ControlNodes".sideTapeAttachment."step".action1[370] )
   END_RUNG
   RUNG wire#w1
      Contact( "Unit1.Em4.ControlNodes".cm.softcam.sideTapeAttachmentAxisY.Pos00_wait.inPos )
      Coil( "Unit1.Em4.ControlNodes".sideTapeAttachment."step".transition1[370] )
   END_RUNG
   RUNG wire#w1
      Contact( "Unit1.Em4.ControlNodes".sideTapeAttachment."step".transition1[370] )
      { S7_Templates := "time_type := Time" } #statTonTime[370].TON(pt := T#100ms, et =>)
      Move(in := #JOB_3_STEP_80, out1 => "Unit1.Em4.ControlNodes".sideTapeAttachment.sequence.status.nextStep)
   END_RUNG
   // the same network as SCL:
   #_w1 := ("Unit1.Em4.ControlNodes".sideTapeAttachment.sequence.status.currentStep = #JOB_3_STEP_70) AND "Unit1.Em4.ControlNodes".sideTapeAttachment.sequence.status.seqActive;
   "Unit1.Em4.ControlNodes".sideTapeAttachment."step".action1[370] := #_w1 AND NOT "Unit1.Em4.ControlNodes".cm.softcam.sideTapeAttachmentAxisY.Pos00_wait.inPos;
   "Unit1.Em4.ControlNodes".sideTapeAttachment."step".transition1[370] := #_w1 AND "Unit1.Em4.ControlNodes".cm.softcam.sideTapeAttachmentAxisY.Pos00_wait.inPos;
   #statTonTime[370].TON(IN := #_w1 AND "Unit1.Em4.ControlNodes".sideTapeAttachment."step".transition1[370],
                         PT := T#100ms);
   IF #statTonTime[370].Q THEN
       "Unit1.Em4.ControlNodes".sideTapeAttachment.sequence.status.nextStep := #JOB_3_STEP_80;
   END_IF;
END_REGION

REGION Network 47: Step[380] : Side Tape Attachment X-Axis Tape-1 Put Pos
   RUNG wire#powerrail
      { S7_Templates := "SrcType := DInt" } EQ_Contact(in1 := "Unit1.Em4.ControlNodes".sideTapeAttachment.sequence.status.currentStep, in2 := #JOB_3_STEP_80)
      Contact( "Unit1.Em4.ControlNodes".sideTapeAttachment.sequence.status.seqActive )
      wire#w1
      I_Contact( "Unit1.Em4.ControlNodes".cm.softcam.sideTapeAttachmentAxisX.pos03_tape1Put.inPos )
      Coil( "Unit1.Em4.ControlNodes".sideTapeAttachment."step".action1[380] )
   END_RUNG
   RUNG wire#w1
      Contact( "Unit1.Em4.ControlNodes".cm.softcam.sideTapeAttachmentAxisX.pos03_tape1Put.inPos )
      Coil( "Unit1.Em4.ControlNodes".sideTapeAttachment."step".transition1[380] )
   END_RUNG
   RUNG wire#w1
      Contact( "Unit1.Em4.ControlNodes".sideTapeAttachment."step".transition1[380] )
      { S7_Templates := "time_type := Time" } #statTonTime[380].TON(pt := T#100ms, et =>)
      Move(in := #JOB_3_STEP_90, out1 => "Unit1.Em4.ControlNodes".sideTapeAttachment.sequence.status.nextStep)
   END_RUNG
   // the same network as SCL:
   #_w1 := ("Unit1.Em4.ControlNodes".sideTapeAttachment.sequence.status.currentStep = #JOB_3_STEP_80) AND "Unit1.Em4.ControlNodes".sideTapeAttachment.sequence.status.seqActive;
   "Unit1.Em4.ControlNodes".sideTapeAttachment."step".action1[380] := #_w1 AND NOT "Unit1.Em4.ControlNodes".cm.softcam.sideTapeAttachmentAxisX.pos03_tape1Put.inPos;
   "Unit1.Em4.ControlNodes".sideTapeAttachment."step".transition1[380] := #_w1 AND "Unit1.Em4.ControlNodes".cm.softcam.sideTapeAttachmentAxisX.pos03_tape1Put.inPos;
   #statTonTime[380].TON(IN := #_w1 AND "Unit1.Em4.ControlNodes".sideTapeAttachment."step".transition1[380],
                         PT := T#100ms);
   IF #statTonTime[380].Q THEN
       "Unit1.Em4.ControlNodes".sideTapeAttachment.sequence.status.nextStep := #JOB_3_STEP_90;
   END_IF;
END_REGION

REGION Network 48: Step[390] : Job[3] Step End
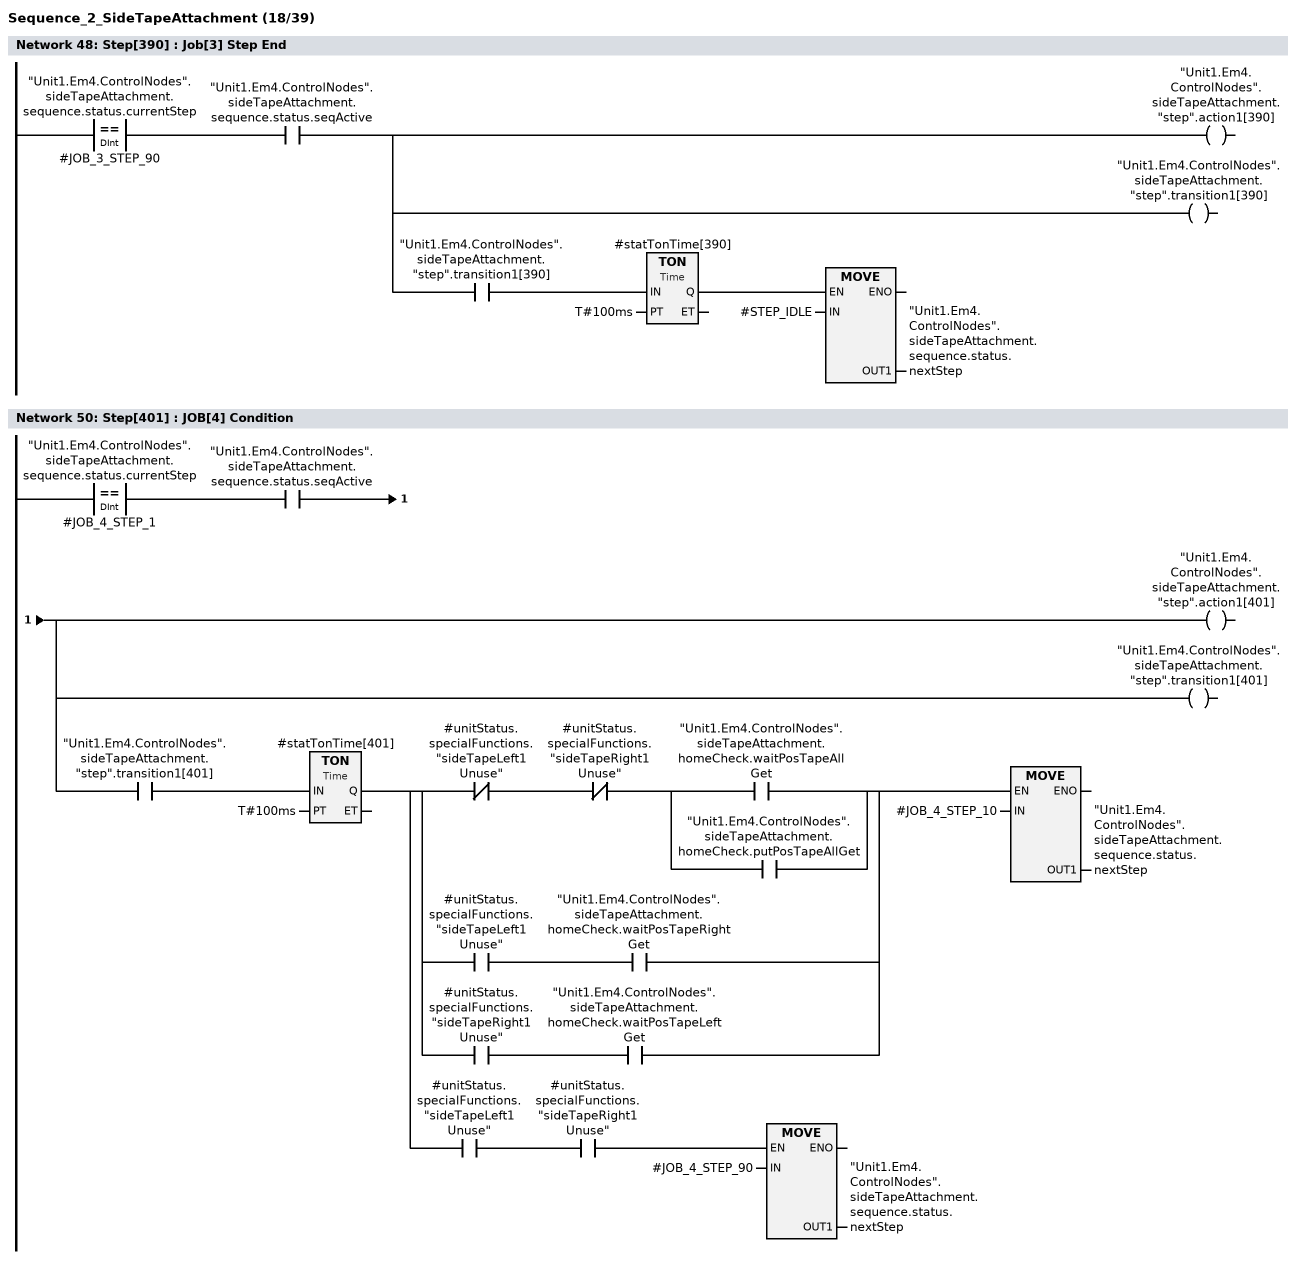
   RUNG wire#powerrail
      { S7_Templates := "SrcType := DInt" } EQ_Contact(in1 := "Unit1.Em4.ControlNodes".sideTapeAttachment.sequence.status.currentStep, in2 := #JOB_3_STEP_90)
      Contact( "Unit1.Em4.ControlNodes".sideTapeAttachment.sequence.status.seqActive )
      wire#w1
      Coil( "Unit1.Em4.ControlNodes".sideTapeAttachment."step".action1[390] )
   END_RUNG
   RUNG wire#w1
      Coil( "Unit1.Em4.ControlNodes".sideTapeAttachment."step".transition1[390] )
   END_RUNG
   RUNG wire#w1
      Contact( "Unit1.Em4.ControlNodes".sideTapeAttachment."step".transition1[390] )
      { S7_Templates := "time_type := Time" } #statTonTime[390].TON(pt := T#100ms, et =>)
      Move(in := #STEP_IDLE, out1 => "Unit1.Em4.ControlNodes".sideTapeAttachment.sequence.status.nextStep)
   END_RUNG
   // the same network as SCL:
   "Unit1.Em4.ControlNodes".sideTapeAttachment."step".action1[390] := ("Unit1.Em4.ControlNodes".sideTapeAttachment.sequence.status.currentStep = #JOB_3_STEP_90) AND "Unit1.Em4.ControlNodes".sideTapeAttachment.sequence.status.seqActive;
   "Unit1.Em4.ControlNodes".sideTapeAttachment."step".transition1[390] := ("Unit1.Em4.ControlNodes".sideTapeAttachment.sequence.status.currentStep = #JOB_3_STEP_90) AND "Unit1.Em4.ControlNodes".sideTapeAttachment.sequence.status.seqActive;
   #statTonTime[390].TON(IN := ("Unit1.Em4.ControlNodes".sideTapeAttachment.sequence.status.currentStep = #JOB_3_STEP_90) AND "Unit1.Em4.ControlNodes".sideTapeAttachment.sequence.status.seqActive AND "Unit1.Em4.ControlNodes".sideTapeAttachment."step".transition1[390],
                         PT := T#100ms);
   IF #statTonTime[390].Q THEN
       "Unit1.Em4.ControlNodes".sideTapeAttachment.sequence.status.nextStep := #STEP_IDLE;
   END_IF;
END_REGION

REGION Network 49: *************** JOB[4] SIDE TAPE PUT-1=AUTO *************************
END_REGION

